LIN {X 0,Y 375.701,Z 668.969,A -85,B 0,C 180,E1 9709.263,E2 9709.263} C_VEL
LIN {X 0,Y 377.557,Z 672.937,A -85,B 0,C 180,E1 9707.734,E2 9707.734} C_VEL
LIN {X 0,Y 377.796,Z 674.692,A -85,B 0,C 180,E1 9707.454,E2 9707.454} C_VEL
LIN {X 0,Y 377.643,Z 677.934,A -85,B 0,C 180,E1 9707.299,E2 9707.299} C_VEL
LIN {X 0,Y 376.937,Z 683.014,A -85,B 0,C 180,E1 9707.331,E2 9707.331} C_VEL
LIN {X 0,Y 374.94,Z 694.139,A -85,B 0,C 180,E1 9707.675,E2 9707.675} C_VEL
LIN {X 0,Y 374.614,Z 696.752,A -85,B 0,C 180,E1 9707.671,E2 9707.671} C_VEL
LIN {X 0,Y 359.205,Z 844.41,A -85,B 0,C 180,E1 9705.429,E2 9705.429} C_VEL
LIN {X 0,Y 354.864,Z 869.774,A -85,B 0,C 180,E1 9704.944,E2 9704.944} C_VEL
LIN {X 0,Y 349.639,Z 892.086,A -85,B 0,C 180,E1 9704.392,E2 9704.392} C_VEL
LIN {X 0,Y 342.832,Z 914.874,A -85,B 0,C 180,E1 9703.649,E2 9703.649} C_VEL
LIN {X 0,Y 335.898,Z 934.267,A -85,B 0,C 180,E1 9702.852,E2 9702.852} C_VEL
LIN {X 0,Y 326.048,Z 957.663,A -85,B 0,C 180,E1 9701.649,E2 9701.649} C_VEL
LIN {X 0,Y 316.768,Z 976.66,A -85,B 0,C 180,E1 9700.43,E2 9700.43} C_VEL
LIN {X 0,Y 304.761,Z 998.24,A -85,B 0,C 180,E1 9698.714,E2 9698.714} C_VEL
LIN {X 0,Y 293.47,Z 1016.27,A -85,B 0,C 180,E1 9696.916,E2 9696.916} C_VEL
LIN {X 0,Y 279.783,Z 1035.844,A -85,B 0,C 180,E1 9694.474,E2 9694.474} C_VEL
LIN {X 0,Y 267.39,Z 1051.959,A -85,B 0,C 180,E1 9691.947,E2 9691.947} C_VEL
LIN {X 0,Y 253.812,Z 1068.099,A -85,B 0,C 180,E1 9688.746,E2 9688.746} C_VEL
LIN {X 0,Y 241.74,Z 1081.488,A -85,B 0,C 180,E1 9685.398,E2 9685.398} C_VEL
LIN {X 0,Y 228.302,Z 1095.466,A -85,B 0,C 180,E1 9680.9,E2 9680.9} C_VEL
LIN {X 0,Y 217.176,Z 1106.587,A -85,B 0,C 180,E1 9676.29,E2 9676.29} C_VEL
LIN {X 0,Y 206.281,Z 1117.208,A -85,B 0,C 180,E1 9670.506,E2 9670.506} C_VEL
LIN {X 0,Y 197.909,Z 1125.557,A -85,B 0,C 180,E1 9664.561,E2 9664.561} C_VEL
LIN {X 0,Y 191.158,Z 1132.65,A -85,B 0,C 180,E1 9657.745,E2 9657.745} C_VEL
LIN {X 0,Y 187.088,Z 1137.624,A -85,B 0,C 180,E1 9651.311,E2 9651.311} C_VEL
LIN {X 0,Y 184.611,Z 1141.644,A -85,B 0,C 180,E1 9643.787,E2 9643.787} C_VEL
LIN {X 0,Y 183.999,Z 1143.579,A -85,B 0,C 180,E1 9637.808,E2 9637.808} C_VEL
LIN {X 0,Y 183.993,Z 1144.393,A -85,B 0,C 180,E1 9632.803,E2 9632.803} C_VEL
LIN {X 0,Y 184.01,Z 1144.46,A -85,B 0,C 180,E1 9628.132,E2 9628.132} C_VEL
LIN {X 0,Y 184,Z 1143.707,A -85,B 0,C 180,E1 9622.82,E2 9622.82} C_VEL
LIN {X 0,Y 184.451,Z 1141.975,A -85,B 0,C 180,E1 9617.158,E2 9617.158} C_VEL
LIN {X 0,Y 186.519,Z 1138.434,A -85,B 0,C 180,E1 9609.935,E2 9609.935} C_VEL
LIN {X 0,Y 190.686,Z 1133.117,A -85,B 0,C 180,E1 9602.858,E2 9602.858} C_VEL
LIN {X 0,Y 197.142,Z 1126.294,A -85,B 0,C 180,E1 9596.088,E2 9596.088} C_VEL
LIN {X 0,Y 205.419,Z 1117.938,A -85,B 0,C 180,E1 9590.02,E2 9590.02} C_VEL
LIN {X 0,Y 215.636,Z 1108.026,A -85,B 0,C 180,E1 9584.431,E2 9584.431} C_VEL
LIN {X 0,Y 227.015,Z 1096.607,A -85,B 0,C 180,E1 9579.575,E2 9579.575} C_VEL
LIN {X 0,Y 239.804,Z 1083.447,A -85,B 0,C 180,E1 9575.19,E2 9575.19} C_VEL
LIN {X 0,Y 252.416,Z 1069.461,A -85,B 0,C 180,E1 9571.605,E2 9571.605} C_VEL
LIN {X 0,Y 265.911,Z 1053.589,A -85,B 0,C 180,E1 9568.369,E2 9568.369} C_VEL
LIN {X 0,Y 278.635,Z 1037.085,A -85,B 0,C 180,E1 9565.735,E2 9565.735} C_VEL
LIN {X 0,Y 291.47,Z 1019.01,A -85,B 0,C 180,E1 9563.413,E2 9563.413} C_VEL
LIN {X 0,Y 303.11,Z 1000.561,A -85,B 0,C 180,E1 9561.525,E2 9561.525} C_VEL
LIN {X 0,Y 314.301,Z 981.008,A -85,B 0,C 180,E1 9559.901,E2 9559.901} C_VEL
LIN {X 0,Y 324.332,Z 960.785,A -85,B 0,C 180,E1 9558.558,E2 9558.558} C_VEL
LIN {X 0,Y 333.728,Z 939.306,A -85,B 0,C 180,E1 9557.394,E2 9557.394} C_VEL
LIN {X 0,Y 341.5,Z 918.015,A -85,B 0,C 180,E1 9556.483,E2 9556.483} C_VEL
LIN {X 0,Y 348.715,Z 894.664,A -85,B 0,C 180,E1 9555.694,E2 9555.694} C_VEL
LIN {X 0,Y 354.348,Z 870.929,A -85,B 0,C 180,E1 9555.095,E2 9555.095} C_VEL
LIN {X 0,Y 358.67,Z 846.5,A -85,B 0,C 180,E1 9554.619,E2 9554.619} C_VEL
LIN {X 0,Y 365.964,Z 777.896,A -85,B 0,C 180,E1 9553.555,E2 9553.555} C_VEL
LIN {X 0,Y 375.97,Z 680.709,A -85,B 0,C 180,E1 9552.089,E2 9552.089} C_VEL
LIN {X 0,Y 373.012,Z 674.26,A -85,B 0,C 180,E1 9549.489,E2 9549.489} C_VEL
LIN {X 0,Y 370.608,Z 669.322,A -85,B 0,C 180,E1 9546.818,E2 9546.818} C_VEL
LIN {X 0,Y 369.056,Z 666.191,A -85,B 0,C 180,E1 9544.506,E2 9544.506} C_VEL
LIN {X 0,Y 367.518,Z 663.322,A -85,B 0,C 180,E1 9540.624,E2 9540.624} C_VEL
LIN {X 0,Y 367.214,Z 663.186,A -85,B 0,C 180,E1 9538.284,E2 9538.284} C_VEL
LIN {X 0,Y 368.066,Z 666.012,A -85,B 0,C 180,E1 9533.605,E2 9533.605} C_VEL
LIN {X 0,Y 369.73,Z 670.596,A -85,B 0,C 180,E1 9530.426,E2 9530.426} C_VEL
LIN {X 0,Y 372.279,Z 677.037,A -85,B 0,C 180,E1 9527.316,E2 9527.316} C_VEL
LIN {X 0,Y 375.214,Z 684.89,A -85,B 0,C 180,E1 9524.564,E2 9524.564} C_VEL
LIN {X 0,Y 358.827,Z 845.607,A -85,B 0,C 180,E1 9522.185,E2 9522.185} C_VEL
LIN {X 0,Y 354.604,Z 870.442,A -85,B 0,C 180,E1 9521.723,E2 9521.723} C_VEL
LIN {X 0,Y 349.339,Z 892.966,A -85,B 0,C 180,E1 9521.175,E2 9521.175} C_VEL
LIN {X 0,Y 342.711,Z 915.03,A -85,B 0,C 180,E1 9520.456,E2 9520.456} C_VEL
LIN {X 0,Y 335.451,Z 935.225,A -85,B 0,C 180,E1 9519.627,E2 9519.627} C_VEL
LIN {X 0,Y 326.046,Z 957.24,A -85,B 0,C 180,E1 9518.487,E2 9518.487} C_VEL
LIN {X 0,Y 317.01,Z 975.595,A -85,B 0,C 180,E1 9517.308,E2 9517.308} C_VEL
LIN {X 0,Y 305.169,Z 996.623,A -85,B 0,C 180,E1 9515.627,E2 9515.627} C_VEL
LIN {X 0,Y 294.024,Z 1014.21,A -85,B 0,C 180,E1 9513.87,E2 9513.87} C_VEL
LIN {X 0,Y 281.274,Z 1032.172,A -85,B 0,C 180,E1 9511.622,E2 9511.622} C_VEL
LIN {X 0,Y 268.993,Z 1047.885,A -85,B 0,C 180,E1 9509.168,E2 9509.168} C_VEL
LIN {X 0,Y 255.516,Z 1063.539,A -85,B 0,C 180,E1 9506.058,E2 9506.058} C_VEL
LIN {X 0,Y 242.86,Z 1077.178,A -85,B 0,C 180,E1 9502.619,E2 9502.619} C_VEL
LIN {X 0,Y 230.542,Z 1089.435,A -85,B 0,C 180,E1 9498.619,E2 9498.619} C_VEL
LIN {X 0,Y 218.914,Z 1100.521,A -85,B 0,C 180,E1 9493.969,E2 9493.969} C_VEL
LIN {X 0,Y 208.319,Z 1110.115,A -85,B 0,C 180,E1 9488.607,E2 9488.607} C_VEL
LIN {X 0,Y 199.344,Z 1118.32,A -85,B 0,C 180,E1 9482.576,E2 9482.576} C_VEL
LIN {X 0,Y 192.297,Z 1124.808,A -85,B 0,C 180,E1 9475.899,E2 9475.899} C_VEL
LIN {X 0,Y 187.614,Z 1129.68,A -85,B 0,C 180,E1 9468.972,E2 9468.972} C_VEL
LIN {X 0,Y 185.097,Z 1132.745,A -85,B 0,C 180,E1 9462.105,E2 9462.105} C_VEL
LIN {X 0,Y 184.194,Z 1134.377,A -85,B 0,C 180,E1 9455.92,E2 9455.92} C_VEL
LIN {X 0,Y 184.04,Z 1134.934,A -85,B 0,C 180,E1 9449.689,E2 9449.689} C_VEL
LIN {X 0,Y 184.237,Z 1134.282,A -85,B 0,C 180,E1 9443.456,E2 9443.456} C_VEL
LIN {X 0,Y 185.163,Z 1132.676,A -85,B 0,C 180,E1 9437.526,E2 9437.526} C_VEL
LIN {X 0,Y 187.925,Z 1129.387,A -85,B 0,C 180,E1 9430.351,E2 9430.351} C_VEL
LIN {X 0,Y 192.747,Z 1124.444,A -85,B 0,C 180,E1 9423.504,E2 9423.504} C_VEL
LIN {X 0,Y 199.846,Z 1117.935,A -85,B 0,C 180,E1 9416.95,E2 9416.95} C_VEL
LIN {X 0,Y 208.659,Z 1109.922,A -85,B 0,C 180,E1 9411.115,E2 9411.115} C_VEL
LIN {X 0,Y 219.841,Z 1099.761,A -85,B 0,C 180,E1 9405.538,E2 9405.538} C_VEL
LIN {X 0,Y 231.005,Z 1089.152,A -85,B 0,C 180,E1 9401.136,E2 9401.136} C_VEL
LIN {X 0,Y 244.665,Z 1075.45,A -85,B 0,C 180,E1 9396.773,E2 9396.773} C_VEL
LIN {X 0,Y 256.763,Z 1062.396,A -85,B 0,C 180,E1 9393.554,E2 9393.554} C_VEL
LIN {X 0,Y 270.582,Z 1046.165,A -85,B 0,C 180,E1 9390.415,E2 9390.415} C_VEL
LIN {X 0,Y 282.352,Z 1031.055,A -85,B 0,C 180,E1 9388.099,E2 9388.099} C_VEL
LIN {X 0,Y 295.457,Z 1012.382,A -85,B 0,C 180,E1 9385.815,E2 9385.815} C_VEL
LIN {X 0,Y 306.65,Z 994.615,A -85,B 0,C 180,E1 9384.077,E2 9384.077} C_VEL
LIN {X 0,Y 318.112,Z 973.95,A -85,B 0,C 180,E1 9382.466,E2 9382.466} C_VEL
LIN {X 0,Y 327.706,Z 954.261,A -85,B 0,C 180,E1 9381.229,E2 9381.229} C_VEL
LIN {X 0,Y 336.673,Z 932.69,A -85,B 0,C 180,E1 9380.152,E2 9380.152} C_VEL
LIN {X 0,Y 343.874,Z 912.39,A -85,B 0,C 180,E1 9379.342,E2 9379.342} C_VEL
LIN {X 0,Y 350.593,Z 889.059,A -85,B 0,C 180,E1 9378.618,E2 9378.618} C_VEL
LIN {X 0,Y 355.597,Z 867.034,A -85,B 0,C 180,E1 9378.102,E2 9378.102} C_VEL
LIN {X 0,Y 359.466,Z 842.639,A -85,B 0,C 180,E1 9377.665,E2 9377.665} C_VEL
LIN {X 0,Y 375.46,Z 685.049,A -85,B 0,C 180,E1 9375.322,E2 9375.322} C_VEL
LIN {X 0,Y 372.379,Z 676.838,A -85,B 0,C 180,E1 9372.405,E2 9372.405} C_VEL
LIN {X 0,Y 369.893,Z 670.489,A -85,B 0,C 180,E1 9369.256,E2 9369.256} C_VEL
LIN {X 0,Y 368.194,Z 665.764,A -85,B 0,C 180,E1 9365.767,E2 9365.767} C_VEL
LIN {X 0,Y 367.559,Z 663.495,A -85,B 0,C 180,E1 9361.091,E2 9361.091} C_VEL
LIN {X 0,Y 368.011,Z 664.084,A -85,B 0,C 180,E1 9358.599,E2 9358.599} C_VEL
LIN {X 0,Y 369.718,Z 667.153,A -85,B 0,C 180,E1 9354.88,E2 9354.88} C_VEL
LIN {X 0,Y 371.838,Z 671.522,A -85,B 0,C 180,E1 9352.04,E2 9352.04} C_VEL
LIN {X 0,Y 374.332,Z 676.68,A -85,B 0,C 180,E1 9349.535,E2 9349.535} C_VEL
LIN {X 0,Y 376.229,Z 681.199,A -85,B 0,C 180,E1 9347.901,E2 9347.901} C_VEL
LIN {X 0,Y 374.614,Z 696.752,A -85,B 0,C 180,E1 9347.671,E2 9347.671} C_VEL
LIN {X 0,Y 373.569,Z 704.446,A -85,B 0,C 180,E1 9347.707,E2 9347.707} C_VEL
LIN {X 0,Y 369.939,Z 724.972,A -85,B 0,C 180,E1 9348.345,E2 9348.345} C_VEL
LIN {X 0,Y 369.073,Z 731.573,A -85,B 0,C 180,E1 9348.36,E2 9348.36} C_VEL
LIN {X 0,Y 357.006,Z 844.853,A -85,B 0,C 180,E1 9346.658,E2 9346.658} C_VEL
LIN {X 0,Y 352.627,Z 869.936,A -85,B 0,C 180,E1 9346.19,E2 9346.19} C_VEL
LIN {X 0,Y 347.283,Z 892.401,A -85,B 0,C 180,E1 9345.649,E2 9345.649} C_VEL
LIN {X 0,Y 340.08,Z 915.965,A -85,B 0,C 180,E1 9344.898,E2 9344.898} C_VEL
LIN {X 0,Y 332.72,Z 936.065,A -85,B 0,C 180,E1 9344.085,E2 9344.085} C_VEL
LIN {X 0,Y 323.145,Z 958.179,A -85,B 0,C 180,E1 9342.965,E2 9342.965} C_VEL
LIN {X 0,Y 313.279,Z 977.938,A -85,B 0,C 180,E1 9341.72,E2 9341.72} C_VEL
LIN {X 0,Y 301.054,Z 999.277,A -85,B 0,C 180,E1 9340.04,E2 9340.04} C_VEL
LIN {X 0,Y 289.54,Z 1017.204,A -85,B 0,C 180,E1 9338.274,E2 9338.274} C_VEL
LIN {X 0,Y 275.944,Z 1036.087,A -85,B 0,C 180,E1 9335.942,E2 9335.942} C_VEL
LIN {X 0,Y 263.611,Z 1051.698,A -85,B 0,C 180,E1 9333.53,E2 9333.53} C_VEL
LIN {X 0,Y 249.62,Z 1067.856,A -85,B 0,C 180,E1 9330.369,E2 9330.369} C_VEL
LIN {X 0,Y 237.131,Z 1081.249,A -85,B 0,C 180,E1 9327.046,E2 9327.046} C_VEL
LIN {X 0,Y 223.656,Z 1094.763,A -85,B 0,C 180,E1 9322.729,E2 9322.729} C_VEL
LIN {X 0,Y 212.066,Z 1105.833,A -85,B 0,C 180,E1 9318.157,E2 9318.157} C_VEL
LIN {X 0,Y 200.5,Z 1116.571,A -85,B 0,C 180,E1 9312.318,E2 9312.318} C_VEL
LIN {X 0,Y 191.77,Z 1124.712,A -85,B 0,C 180,E1 9306.47,E2 9306.47} C_VEL
LIN {X 0,Y 184.148,Z 1132.17,A -85,B 0,C 180,E1 9299.254,E2 9299.254} C_VEL
LIN {X 0,Y 179.628,Z 1137.193,A -85,B 0,C 180,E1 9292.587,E2 9292.587} C_VEL
LIN {X 0,Y 176.786,Z 1141.319,A -85,B 0,C 180,E1 9284.722,E2 9284.722} C_VEL
LIN {X 0,Y 176.01,Z 1143.368,A -85,B 0,C 180,E1 9278.165,E2 9278.165} C_VEL
LIN {X 0,Y 175.994,Z 1144.183,A -85,B 0,C 180,E1 9272.931,E2 9272.931} C_VEL
LIN {X 0,Y 176.01,Z 1144.25,A -85,B 0,C 180,E1 9268.047,E2 9268.047} C_VEL
LIN {X 0,Y 176.001,Z 1143.568,A -85,B 0,C 180,E1 9262.82,E2 9262.82} C_VEL
LIN {X 0,Y 176.481,Z 1141.881,A -85,B 0,C 180,E1 9256.901,E2 9256.901} C_VEL
LIN {X 0,Y 178.418,Z 1138.742,A -85,B 0,C 180,E1 9250.01,E2 9250.01} C_VEL
LIN {X 0,Y 182.894,Z 1133.424,A -85,B 0,C 180,E1 9242.309,E2 9242.309} C_VEL
LIN {X 0,Y 188.94,Z 1127.333,A -85,B 0,C 180,E1 9235.877,E2 9235.877} C_VEL
LIN {X 0,Y 198.247,Z 1118.544,A -85,B 0,C 180,E1 9229.029,E2 9229.029} C_VEL
LIN {X 0,Y 207.807,Z 1109.679,A -85,B 0,C 180,E1 9223.801,E2 9223.801} C_VEL
LIN {X 0,Y 220.623,Z 1097.543,A -85,B 0,C 180,E1 9218.366,E2 9218.366} C_VEL
LIN {X 0,Y 232.489,Z 1085.818,A -85,B 0,C 180,E1 9214.334,E2 9214.334} C_VEL
LIN {X 0,Y 246.765,Z 1070.777,A -85,B 0,C 180,E1 9210.336,E2 9210.336} C_VEL
LIN {X 0,Y 259.098,Z 1056.809,A -85,B 0,C 180,E1 9207.427,E2 9207.427} C_VEL
LIN {X 0,Y 273.581,Z 1038.886,A -85,B 0,C 180,E1 9204.487,E2 9204.487} C_VEL
LIN {X 0,Y 285.48,Z 1022.721,A -85,B 0,C 180,E1 9202.383,E2 9202.383} C_VEL
LIN {X 0,Y 298.547,Z 1002.939,A -85,B 0,C 180,E1 9200.318,E2 9200.318} C_VEL
LIN {X 0,Y 309.019,Z 985.235,A -85,B 0,C 180,E1 9198.836,E2 9198.836} C_VEL
LIN {X 0,Y 320.542,Z 963.106,A -85,B 0,C 180,E1 9197.343,E2 9197.343} C_VEL
LIN {X 0,Y 329.2,Z 943.943,A -85,B 0,C 180,E1 9196.3,E2 9196.3} C_VEL
LIN {X 0,Y 338.406,Z 920.041,A -85,B 0,C 180,E1 9195.265,E2 9195.265} C_VEL
LIN {X 0,Y 345.052,Z 899.254,A -85,B 0,C 180,E1 9194.564,E2 9194.564} C_VEL
LIN {X 0,Y 351.521,Z 873.81,A -85,B 0,C 180,E1 9193.908,E2 9193.908} C_VEL
LIN {X 0,Y 355.776,Z 851.301,A -85,B 0,C 180,E1 9193.466,E2 9193.466} C_VEL
LIN {X 0,Y 359.782,Z 817.87,A -85,B 0,C 180,E1 9192.936,E2 9192.936} C_VEL
LIN {X 0,Y 373.543,Z 686.091,A -85,B 0,C 180,E1 9190.956,E2 9190.956} C_VEL
LIN {X 0,Y 370.614,Z 679.643,A -85,B 0,C 180,E1 9188.065,E2 9188.065} C_VEL
LIN {X 0,Y 369.036,Z 676.353,A -85,B 0,C 180,E1 9186.066,E2 9186.066} C_VEL
LIN {X 0,Y 367.984,Z 674.066,A -85,B 0,C 180,E1 9184.363,E2 9184.363} C_VEL
LIN {X 0,Y 366.509,Z 671.213,A -85,B 0,C 180,E1 9180.469,E2 9180.469} C_VEL
LIN {X 0,Y 366.233,Z 671.188,A -85,B 0,C 180,E1 9178.122,E2 9178.122} C_VEL
LIN {X 0,Y 367.02,Z 673.937,A -85,B 0,C 180,E1 9173.744,E2 9173.744} C_VEL
LIN {X 0,Y 368.587,Z 678.422,A -85,B 0,C 180,E1 9170.632,E2 9170.632} C_VEL
LIN {X 0,Y 370.912,Z 684.617,A -85,B 0,C 180,E1 9167.664,E2 9167.664} C_VEL
LIN {X 0,Y 372.841,Z 690.31,A -85,B 0,C 180,E1 9165.682,E2 9165.682} C_VEL
LIN {X 0,Y 356.687,Z 845.48,A -85,B 0,C 180,E1 9163.423,E2 9163.423} C_VEL
LIN {X 0,Y 352.383,Z 870.437,A -85,B 0,C 180,E1 9162.971,E2 9162.971} C_VEL
LIN {X 0,Y 347.07,Z 892.849,A -85,B 0,C 180,E1 9162.443,E2 9162.443} C_VEL
LIN {X 0,Y 340.123,Z 915.582,A -85,B 0,C 180,E1 9161.724,E2 9161.724} C_VEL
LIN {X 0,Y 332.752,Z 935.713,A -85,B 0,C 180,E1 9160.918,E2 9160.918} C_VEL
LIN {X 0,Y 323.453,Z 957.092,A -85,B 0,C 180,E1 9159.84,E2 9159.84} C_VEL
LIN {X 0,Y 313.999,Z 975.96,A -85,B 0,C 180,E1 9158.659,E2 9158.659} C_VEL
LIN {X 0,Y 301.936,Z 996.938,A -85,B 0,C 180,E1 9157.018,E2 9157.018} C_VEL
LIN {X 0,Y 290.559,Z 1014.508,A -85,B 0,C 180,E1 9155.299,E2 9155.299} C_VEL
LIN {X 0,Y 277.52,Z 1032.443,A -85,B 0,C 180,E1 9153.092,E2 9153.092} C_VEL
LIN {X 0,Y 264.928,Z 1048.146,A -85,B 0,C 180,E1 9150.674,E2 9150.674} C_VEL
LIN {X 0,Y 251.069,Z 1063.785,A -85,B 0,C 180,E1 9147.597,E2 9147.597} C_VEL
LIN {X 0,Y 238.007,Z 1077.418,A -85,B 0,C 180,E1 9144.176,E2 9144.176} C_VEL
LIN {X 0,Y 225.235,Z 1089.663,A -85,B 0,C 180,E1 9140.175,E2 9140.175} C_VEL
LIN {X 0,Y 213.657,Z 1100.242,A -85,B 0,C 180,E1 9135.728,E2 9135.728} C_VEL
LIN {X 0,Y 202.468,Z 1109.939,A -85,B 0,C 180,E1 9130.312,E2 9130.312} C_VEL
LIN {X 0,Y 193.141,Z 1117.975,A -85,B 0,C 180,E1 9124.353,E2 9124.353} C_VEL
LIN {X 0,Y 185.556,Z 1124.53,A -85,B 0,C 180,E1 9117.608,E2 9117.608} C_VEL
LIN {X 0,Y 180.308,Z 1129.536,A -85,B 0,C 180,E1 9110.448,E2 9110.448} C_VEL
LIN {X 0,Y 177.312,Z 1132.828,A -85,B 0,C 180,E1 9103.036,E2 9103.036} C_VEL
LIN {X 0,Y 176.266,Z 1134.457,A -85,B 0,C 180,E1 9096.842,E2 9096.842} C_VEL
LIN {X 0,Y 176.047,Z 1135.132,A -85,B 0,C 180,E1 9090.325,E2 9090.325} C_VEL
LIN {X 0,Y 176.21,Z 1134.623,A -85,B 0,C 180,E1 9083.811,E2 9083.811} C_VEL
LIN {X 0,Y 177.205,Z 1132.996,A -85,B 0,C 180,E1 9077.287,E2 9077.287} C_VEL
LIN {X 0,Y 180.089,Z 1129.82,A -85,B 0,C 180,E1 9069.865,E2 9069.865} C_VEL
LIN {X 0,Y 185.214,Z 1124.905,A -85,B 0,C 180,E1 9062.685,E2 9062.685} C_VEL
LIN {X 0,Y 192.679,Z 1118.493,A -85,B 0,C 180,E1 9055.912,E2 9055.912} C_VEL
LIN {X 0,Y 202.365,Z 1110.14,A -85,B 0,C 180,E1 9049.663,E2 9049.663} C_VEL
LIN {X 0,Y 214.088,Z 1099.984,A -85,B 0,C 180,E1 9044.007,E2 9044.007} C_VEL
LIN {X 0,Y 225.724,Z 1089.376,A -85,B 0,C 180,E1 9039.577,E2 9039.577} C_VEL
LIN {X 0,Y 239.88,Z 1075.684,A -85,B 0,C 180,E1 9035.215,E2 9035.215} C_VEL
LIN {X 0,Y 252.36,Z 1062.634,A -85,B 0,C 180,E1 9032.015,E2 9032.015} C_VEL
LIN {X 0,Y 266.293,Z 1046.756,A -85,B 0,C 180,E1 9028.969,E2 9028.969} C_VEL
LIN {X 0,Y 278.555,Z 1031.418,A -85,B 0,C 180,E1 9026.645,E2 9026.645} C_VEL
LIN {X 0,Y 292.033,Z 1012.673,A -85,B 0,C 180,E1 9024.389,E2 9024.389} C_VEL
LIN {X 0,Y 303.454,Z 994.922,A -85,B 0,C 180,E1 9022.689,E2 9022.689} C_VEL
LIN {X 0,Y 315.131,Z 974.305,A -85,B 0,C 180,E1 9021.117,E2 9021.117} C_VEL
LIN {X 0,Y 324.889,Z 954.646,A -85,B 0,C 180,E1 9019.911,E2 9019.911} C_VEL
LIN {X 0,Y 334.014,Z 933.135,A -85,B 0,C 180,E1 9018.863,E2 9018.863} C_VEL
LIN {X 0,Y 341.269,Z 913.053,A -85,B 0,C 180,E1 9018.081,E2 9018.081} C_VEL
LIN {X 0,Y 348.28,Z 889.203,A -85,B 0,C 180,E1 9017.36,E2 9017.36} C_VEL
LIN {X 0,Y 353.371,Z 867.137,A -85,B 0,C 180,E1 9016.859,E2 9016.859} C_VEL
LIN {X 0,Y 357.33,Z 842.607,A -85,B 0,C 180,E1 9016.429,E2 9016.429} C_VEL
LIN {X 0,Y 373.1,Z 690.229,A -85,B 0,C 180,E1 9014.195,E2 9014.195} C_VEL
LIN {X 0,Y 370.431,Z 682.823,A -85,B 0,C 180,E1 9011.364,E2 9011.364} C_VEL
LIN {X 0,Y 368.48,Z 677.548,A -85,B 0,C 180,E1 9008.583,E2 9008.583} C_VEL
LIN {X 0,Y 367.113,Z 673.554,A -85,B 0,C 180,E1 9005.47,E2 9005.47} C_VEL
LIN {X 0,Y 366.583,Z 671.437,A -85,B 0,C 180,E1 9001.094,E2 9001.094} C_VEL
LIN {X 0,Y 367.023,Z 672.068,A -85,B 0,C 180,E1 8998.595,E2 8998.595} C_VEL
LIN {X 0,Y 368.625,Z 675.066,A -85,B 0,C 180,E1 8995.02,E2 8995.02} C_VEL
LIN {X 0,Y 370.568,Z 679.204,A -85,B 0,C 180,E1 8992.324,E2 8992.324} C_VEL
LIN {X 0,Y 372.89,Z 684.225,A -85,B 0,C 180,E1 8989.884,E2 8989.884} C_VEL
LIN {X 0,Y 373.813,Z 686.677,A -85,B 0,C 180,E1 8989.013,E2 8989.013} C_VEL
LIN {X 0,Y 369.073,Z 731.573,A -85,B 0,C 180,E1 8988.36,E2 8988.36} C_VEL
LIN {X 0,Y 368.033,Z 739.267,A -85,B 0,C 180,E1 8988.399,E2 8988.399} C_VEL
LIN {X 0,Y 364.446,Z 759.789,A -85,B 0,C 180,E1 8989.058,E2 8989.058} C_VEL
LIN {X 0,Y 363.586,Z 766.389,A -85,B 0,C 180,E1 8989.073,E2 8989.073} C_VEL
LIN {X 0,Y 354.933,Z 845.615,A -85,B 0,C 180,E1 8987.896,E2 8987.896} C_VEL
LIN {X 0,Y 350.516,Z 870.293,A -85,B 0,C 180,E1 8987.446,E2 8987.446} C_VEL
LIN {X 0,Y 344.987,Z 893.137,A -85,B 0,C 180,E1 8986.912,E2 8986.912} C_VEL
LIN {X 0,Y 337.729,Z 916.376,A -85,B 0,C 180,E1 8986.19,E2 8986.19} C_VEL
LIN {X 0,Y 329.699,Z 937.863,A -85,B 0,C 180,E1 8985.341,E2 8985.341} C_VEL
LIN {X 0,Y 319.977,Z 959.603,A -85,B 0,C 180,E1 8984.253,E2 8984.253} C_VEL
LIN {X 0,Y 309.522,Z 980.035,A -85,B 0,C 180,E1 8982.982,E2 8982.982} C_VEL
LIN {X 0,Y 297.511,Z 1000.314,A -85,B 0,C 180,E1 8981.399,E2 8981.399} C_VEL
LIN {X 0,Y 284.95,Z 1019.364,A -85,B 0,C 180,E1 8979.538,E2 8979.538} C_VEL
LIN {X 0,Y 271.489,Z 1037.358,A -85,B 0,C 180,E1 8977.308,E2 8977.308} C_VEL
LIN {X 0,Y 257.723,Z 1054.217,A -85,B 0,C 180,E1 8974.686,E2 8974.686} C_VEL
LIN {X 0,Y 243.646,Z 1069.732,A -85,B 0,C 180,E1 8971.572,E2 8971.572} C_VEL
LIN {X 0,Y 229.291,Z 1084.458,A -85,B 0,C 180,E1 8967.779,E2 8967.779} C_VEL
LIN {X 0,Y 216.208,Z 1096.873,A -85,B 0,C 180,E1 8963.581,E2 8963.581} C_VEL
LIN {X 0,Y 203.194,Z 1108.679,A -85,B 0,C 180,E1 8958.37,E2 8958.37} C_VEL
LIN {X 0,Y 192.535,Z 1118.01,A -85,B 0,C 180,E1 8952.869,E2 8952.869} C_VEL
LIN {X 0,Y 182.883,Z 1126.566,A -85,B 0,C 180,E1 8946.191,E2 8946.191} C_VEL
LIN {X 0,Y 175.894,Z 1133.006,A -85,B 0,C 180,E1 8939.267,E2 8939.267} C_VEL
LIN {X 0,Y 171.05,Z 1138.232,A -85,B 0,C 180,E1 8931.609,E2 8931.609} C_VEL
LIN {X 0,Y 168.635,Z 1141.576,A -85,B 0,C 180,E1 8924.07,E2 8924.07} C_VEL
LIN {X 0,Y 168.002,Z 1143.301,A -85,B 0,C 180,E1 8917.868,E2 8917.868} C_VEL
LIN {X 0,Y 168.004,Z 1144.021,A -85,B 0,C 180,E1 8912.388,E2 8912.388} C_VEL
LIN {X 0,Y 168.004,Z 1144.016,A -85,B 0,C 180,E1 8907.612,E2 8907.612} C_VEL
LIN {X 0,Y 168.005,Z 1143.284,A -85,B 0,C 180,E1 8902.132,E2 8902.132} C_VEL
LIN {X 0,Y 168.635,Z 1141.548,A -85,B 0,C 180,E1 8895.93,E2 8895.93} C_VEL
LIN {X 0,Y 171.208,Z 1137.999,A -85,B 0,C 180,E1 8888.051,E2 8888.051} C_VEL
LIN {X 0,Y 176.157,Z 1132.678,A -85,B 0,C 180,E1 8880.408,E2 8880.408} C_VEL
LIN {X 0,Y 183.692,Z 1125.785,A -85,B 0,C 180,E1 8873.146,E2 8873.146} C_VEL
LIN {X 0,Y 193.472,Z 1117.075,A -85,B 0,C 180,E1 8866.578,E2 8866.578} C_VEL
LIN {X 0,Y 205.033,Z 1106.942,A -85,B 0,C 180,E1 8860.805,E2 8860.805} C_VEL
LIN {X 0,Y 217.45,Z 1095.554,A -85,B 0,C 180,E1 8855.973,E2 8855.973} C_VEL
LIN {X 0,Y 231.332,Z 1082.246,A -85,B 0,C 180,E1 8851.624,E2 8851.624} C_VEL
LIN {X 0,Y 244.885,Z 1068.18,A -85,B 0,C 180,E1 8848.121,E2 8848.121} C_VEL
LIN {X 0,Y 259.249,Z 1052.117,A -85,B 0,C 180,E1 8844.991,E2 8844.991} C_VEL
LIN {X 0,Y 272.217,Z 1036.117,A -85,B 0,C 180,E1 8842.552,E2 8842.552} C_VEL
LIN {X 0,Y 285.758,Z 1017.785,A -85,B 0,C 180,E1 8840.322,E2 8840.322} C_VEL
LIN {X 0,Y 297.492,Z 999.917,A -85,B 0,C 180,E1 8838.59,E2 8838.59} C_VEL
LIN {X 0,Y 309.502,Z 979.549,A -85,B 0,C 180,E1 8837.006,E2 8837.006} C_VEL
LIN {X 0,Y 319.655,Z 959.701,A -85,B 0,C 180,E1 8835.771,E2 8835.771} C_VEL
LIN {X 0,Y 329.205,Z 938.415,A -85,B 0,C 180,E1 8834.699,E2 8834.699} C_VEL
LIN {X 0,Y 337.262,Z 916.897,A -85,B 0,C 180,E1 8833.843,E2 8833.843} C_VEL
LIN {X 0,Y 344.576,Z 893.611,A -85,B 0,C 180,E1 8833.114,E2 8833.114} C_VEL
LIN {X 0,Y 350.172,Z 870.54,A -85,B 0,C 180,E1 8832.571,E2 8832.571} C_VEL
LIN {X 0,Y 354.603,Z 845.902,A -85,B 0,C 180,E1 8832.121,E2 8832.121} C_VEL
LIN {X 0,Y 363.543,Z 764.207,A -85,B 0,C 180,E1 8830.905,E2 8830.905} C_VEL
LIN {X 0,Y 371.28,Z 691.711,A -85,B 0,C 180,E1 8829.847,E2 8829.847} C_VEL
LIN {X 0,Y 368.831,Z 686.149,A -85,B 0,C 180,E1 8827.151,E2 8827.151} C_VEL
LIN {X 0,Y 366.915,Z 681.941,A -85,B 0,C 180,E1 8824.22,E2 8824.22} C_VEL
LIN {X 0,Y 365.502,Z 679.106,A -85,B 0,C 180,E1 8820.313,E2 8820.313} C_VEL
LIN {X 0,Y 365.252,Z 679.205,A -85,B 0,C 180,E1 8817.961,E2 8817.961} C_VEL
LIN {X 0,Y 365.976,Z 681.858,A -85,B 0,C 180,E1 8813.883,E2 8813.883} C_VEL
LIN {X 0,Y 367.448,Z 686.247,A -85,B 0,C 180,E1 8810.84,E2 8810.84} C_VEL
LIN {X 0,Y 369.555,Z 692.195,A -85,B 0,C 180,E1 8808.015,E2 8808.015} C_VEL
LIN {X 0,Y 370.623,Z 695.601,A -85,B 0,C 180,E1 8806.815,E2 8806.815} C_VEL
LIN {X 0,Y 354.676,Z 845.674,A -85,B 0,C 180,E1 8804.671,E2 8804.671} C_VEL
LIN {X 0,Y 350.33,Z 870.434,A -85,B 0,C 180,E1 8804.235,E2 8804.235} C_VEL
LIN {X 0,Y 344.945,Z 892.839,A -85,B 0,C 180,E1 8803.725,E2 8803.725} C_VEL
LIN {X 0,Y 337.705,Z 916.132,A -85,B 0,C 180,E1 8803.01,E2 8803.01} C_VEL
LIN {X 0,Y 329.547,Z 937.943,A -85,B 0,C 180,E1 8802.155,E2 8802.155} C_VEL
LIN {X 0,Y 320.201,Z 958.683,A -85,B 0,C 180,E1 8801.117,E2 8801.117} C_VEL
LIN {X 0,Y 309.892,Z 978.739,A -85,B 0,C 180,E1 8799.874,E2 8799.874} C_VEL
LIN {X 0,Y 298.376,Z 998.057,A -85,B 0,C 180,E1 8798.369,E2 8798.369} C_VEL
LIN {X 0,Y 286.059,Z 1016.613,A -85,B 0,C 180,E1 8796.57,E2 8796.57} C_VEL
LIN {X 0,Y 272.763,Z 1034.215,A -85,B 0,C 180,E1 8794.394,E2 8794.394} C_VEL
LIN {X 0,Y 259.527,Z 1050.22,A -85,B 0,C 180,E1 8791.919,E2 8791.919} C_VEL
LIN {X 0,Y 246.081,Z 1064.788,A -85,B 0,C 180,E1 8789.021,E2 8789.021} C_VEL
LIN {X 0,Y 232.652,Z 1078.344,A -85,B 0,C 180,E1 8785.607,E2 8785.607} C_VEL
LIN {X 0,Y 219.469,Z 1090.457,A -85,B 0,C 180,E1 8781.594,E2 8781.594} C_VEL
LIN {X 0,Y 206.908,Z 1101.471,A -85,B 0,C 180,E1 8776.863,E2 8776.863} C_VEL
LIN {X 0,Y 195.334,Z 1110.951,A -85,B 0,C 180,E1 8771.326,E2 8771.326} C_VEL
LIN {X 0,Y 185.227,Z 1119.189,A -85,B 0,C 180,E1 8764.862,E2 8764.862} C_VEL
LIN {X 0,Y 177.786,Z 1125.24,A -85,B 0,C 180,E1 8758.192,E2 8758.192} C_VEL
LIN {X 0,Y 172.346,Z 1130.106,A -85,B 0,C 180,E1 8750.726,E2 8750.726} C_VEL
LIN {X 0,Y 169.362,Z 1133.15,A -85,B 0,C 180,E1 8743.312,E2 8743.312} C_VEL
LIN {X 0,Y 168.238,Z 1134.799,A -85,B 0,C 180,E1 8736.484,E2 8736.484} C_VEL
LIN {X 0,Y 168.045,Z 1135.354,A -85,B 0,C 180,E1 8729.659,E2 8729.659} C_VEL
LIN {X 0,Y 168.293,Z 1134.703,A -85,B 0,C 180,E1 8722.833,E2 8722.833} C_VEL
LIN {X 0,Y 169.431,Z 1133.099,A -85,B 0,C 180,E1 8716.346,E2 8716.346} C_VEL
LIN {X 0,Y 172.68,Z 1129.854,A -85,B 0,C 180,E1 8708.605,E2 8708.605} C_VEL
LIN {X 0,Y 178.308,Z 1124.872,A -85,B 0,C 180,E1 8701.167,E2 8701.167} C_VEL
LIN {X 0,Y 186.373,Z 1118.37,A -85,B 0,C 180,E1 8694.212,E2 8694.212} C_VEL
LIN {X 0,Y 196.418,Z 1110.19,A -85,B 0,C 180,E1 8688.008,E2 8688.008} C_VEL
LIN {X 0,Y 208.497,Z 1100.207,A -85,B 0,C 180,E1 8682.393,E2 8682.393} C_VEL
LIN {X 0,Y 220.619,Z 1089.6,A -85,B 0,C 180,E1 8677.944,E2 8677.944} C_VEL
LIN {X 0,Y 235.279,Z 1075.917,A -85,B 0,C 180,E1 8673.595,E2 8673.595} C_VEL
LIN {X 0,Y 248.146,Z 1062.874,A -85,B 0,C 180,E1 8670.423,E2 8670.423} C_VEL
LIN {X 0,Y 262.461,Z 1047.011,A -85,B 0,C 180,E1 8667.42,E2 8667.42} C_VEL
LIN {X 0,Y 275.022,Z 1031.681,A -85,B 0,C 180,E1 8665.138,E2 8665.138} C_VEL
LIN {X 0,Y 289.075,Z 1012.552,A -85,B 0,C 180,E1 8662.889,E2 8662.889} C_VEL
LIN {X 0,Y 300.82,Z 994.633,A -85,B 0,C 180,E1 8661.221,E2 8661.221} C_VEL
LIN {X 0,Y 312.328,Z 974.659,A -85,B 0,C 180,E1 8659.742,E2 8659.742} C_VEL
LIN {X 0,Y 322.248,Z 955.031,A -85,B 0,C 180,E1 8658.571,E2 8658.571} C_VEL
LIN {X 0,Y 331.815,Z 932.84,A -85,B 0,C 180,E1 8657.523,E2 8657.523} C_VEL
LIN {X 0,Y 339.365,Z 912.181,A -85,B 0,C 180,E1 8656.75,E2 8656.75} C_VEL
LIN {X 0,Y 346.282,Z 888.782,A -85,B 0,C 180,E1 8656.073,E2 8656.073} C_VEL
LIN {X 0,Y 351.481,Z 866.456,A -85,B 0,C 180,E1 8655.585,E2 8655.585} C_VEL
LIN {X 0,Y 355.411,Z 842.166,A -85,B 0,C 180,E1 8655.174,E2 8655.174} C_VEL
LIN {X 0,Y 370.892,Z 695.586,A -85,B 0,C 180,E1 8653.069,E2 8653.069} C_VEL
LIN {X 0,Y 368.931,Z 689.932,A -85,B 0,C 180,E1 8650.778,E2 8650.778} C_VEL
LIN {X 0,Y 367.277,Z 685.115,A -85,B 0,C 180,E1 8648.217,E2 8648.217} C_VEL
LIN {X 0,Y 366.093,Z 681.44,A -85,B 0,C 180,E1 8645.328,E2 8645.328} C_VEL
LIN {X 0,Y 365.608,Z 679.379,A -85,B 0,C 180,E1 8641.097,E2 8641.097} C_VEL
LIN {X 0,Y 365.996,Z 679.944,A -85,B 0,C 180,E1 8638.748,E2 8638.748} C_VEL
LIN {X 0,Y 367.491,Z 682.864,A -85,B 0,C 180,E1 8635.24,E2 8635.24} C_VEL
LIN {X 0,Y 369.304,Z 686.886,A -85,B 0,C 180,E1 8632.611,E2 8632.611} C_VEL
LIN {X 0,Y 371.556,Z 692.01,A -85,B 0,C 180,E1 8630.142,E2 8630.142} C_VEL
LIN {X 0,Y 363.586,Z 766.389,A -85,B 0,C 180,E1 8629.073,E2 8629.073} C_VEL
LIN {X 0,Y 362.56,Z 774.081,A -85,B 0,C 180,E1 8629.109,E2 8629.109} C_VEL
LIN {X 0,Y 359.045,Z 794.605,A -85,B 0,C 180,E1 8629.789,E2 8629.789} C_VEL
LIN {X 0,Y 358.183,Z 801.208,A -85,B 0,C 180,E1 8629.811,E2 8629.811} C_VEL
LIN {X 0,Y 352.747,Z 848.47,A -85,B 0,C 180,E1 8629.116,E2 8629.116} C_VEL
LIN {X 0,Y 348.203,Z 872.349,A -85,B 0,C 180,E1 8628.683,E2 8628.683} C_VEL
LIN {X 0,Y 342.274,Z 895.904,A -85,B 0,C 180,E1 8628.138,E2 8628.138} C_VEL
LIN {X 0,Y 334.976,Z 918.42,A -85,B 0,C 180,E1 8627.445,E2 8627.445} C_VEL
LIN {X 0,Y 326.385,Z 940.628,A -85,B 0,C 180,E1 8626.575,E2 8626.575} C_VEL
LIN {X 0,Y 316.974,Z 961.028,A -85,B 0,C 180,E1 8625.565,E2 8625.565} C_VEL
LIN {X 0,Y 305.871,Z 982.105,A -85,B 0,C 180,E1 8624.272,E2 8624.272} C_VEL
LIN {X 0,Y 294.14,Z 1001.349,A -85,B 0,C 180,E1 8622.79,E2 8622.79} C_VEL
LIN {X 0,Y 281.342,Z 1020.227,A -85,B 0,C 180,E1 8620.974,E2 8620.974} C_VEL
LIN {X 0,Y 268.012,Z 1037.603,A -85,B 0,C 180,E1 8618.859,E2 8618.859} C_VEL
LIN {X 0,Y 253.513,Z 1054.825,A -85,B 0,C 180,E1 8616.212,E2 8616.212} C_VEL
LIN {X 0,Y 239.601,Z 1069.714,A -85,B 0,C 180,E1 8613.26,E2 8613.26} C_VEL
LIN {X 0,Y 224.925,Z 1084.276,A -85,B 0,C 180,E1 8609.55,E2 8609.55} C_VEL
LIN {X 0,Y 211.386,Z 1096.643,A -85,B 0,C 180,E1 8605.391,E2 8605.391} C_VEL
LIN {X 0,Y 197.838,Z 1108.406,A -85,B 0,C 180,E1 8600.195,E2 8600.195} C_VEL
LIN {X 0,Y 186.536,Z 1117.788,A -85,B 0,C 180,E1 8594.604,E2 8594.604} C_VEL
LIN {X 0,Y 175.871,Z 1126.659,A -85,B 0,C 180,E1 8587.469,E2 8587.469} C_VEL
LIN {X 0,Y 168.738,Z 1132.788,A -85,B 0,C 180,E1 8580.638,E2 8580.638} C_VEL
LIN {X 0,Y 163.329,Z 1138.135,A -85,B 0,C 180,E1 8572.42,E2 8572.42} C_VEL
LIN {X 0,Y 160.755,Z 1141.364,A -85,B 0,C 180,E1 8564.775,E2 8564.775} C_VEL
LIN {X 0,Y 160.015,Z 1143.089,A -85,B 0,C 180,E1 8558.263,E2 8558.263} C_VEL
LIN {X 0,Y 160.004,Z 1143.812,A -85,B 0,C 180,E1 8552.507,E2 8552.507} C_VEL
LIN {X 0,Y 160.004,Z 1143.806,A -85,B 0,C 180,E1 8547.493,E2 8547.493} C_VEL
LIN {X 0,Y 160.016,Z 1143.072,A -85,B 0,C 180,E1 8541.737,E2 8541.737} C_VEL
LIN {X 0,Y 160.755,Z 1141.334,A -85,B 0,C 180,E1 8535.225,E2 8535.225} C_VEL
LIN {X 0,Y 163.622,Z 1137.782,A -85,B 0,C 180,E1 8526.977,E2 8526.977} C_VEL
LIN {X 0,Y 169.022,Z 1132.46,A -85,B 0,C 180,E1 8519.024,E2 8519.024} C_VEL
LIN {X 0,Y 177.055,Z 1125.628,A -85,B 0,C 180,E1 8511.595,E2 8511.595} C_VEL
LIN {X 0,Y 187.528,Z 1116.85,A -85,B 0,C 180,E1 8504.834,E2 8504.834} C_VEL
LIN {X 0,Y 199.58,Z 1106.823,A -85,B 0,C 180,E1 8499.054,E2 8499.054} C_VEL
LIN {X 0,Y 212.679,Z 1095.321,A -85,B 0,C 180,E1 8494.162,E2 8494.162} C_VEL
LIN {X 0,Y 227.149,Z 1081.948,A -85,B 0,C 180,E1 8489.829,E2 8489.829} C_VEL
LIN {X 0,Y 240.34,Z 1068.714,A -85,B 0,C 180,E1 8486.559,E2 8486.559} C_VEL
LIN {X 0,Y 255.081,Z 1052.79,A -85,B 0,C 180,E1 8483.471,E2 8483.471} C_VEL
LIN {X 0,Y 268.818,Z 1036.281,A -85,B 0,C 180,E1 8480.994,E2 8480.994} C_VEL
LIN {X 0,Y 282.592,Z 1018.096,A -85,B 0,C 180,E1 8478.827,E2 8478.827} C_VEL
LIN {X 0,Y 294.986,Z 999.596,A -85,B 0,C 180,E1 8477.084,E2 8477.084} C_VEL
LIN {X 0,Y 307.215,Z 979.179,A -85,B 0,C 180,E1 8475.55,E2 8475.55} C_VEL
LIN {X 0,Y 317.402,Z 959.576,A -85,B 0,C 180,E1 8474.372,E2 8474.372} C_VEL
LIN {X 0,Y 327.271,Z 937.838,A -85,B 0,C 180,E1 8473.32,E2 8473.32} C_VEL
LIN {X 0,Y 335.417,Z 916.341,A -85,B 0,C 180,E1 8472.5,E2 8472.5} C_VEL
LIN {X 0,Y 342.866,Z 892.728,A -85,B 0,C 180,E1 8471.794,E2 8471.794} C_VEL
LIN {X 0,Y 348.387,Z 870.155,A -85,B 0,C 180,E1 8471.285,E2 8471.285} C_VEL
LIN {X 0,Y 352.89,Z 845.122,A -85,B 0,C 180,E1 8470.844,E2 8470.844} C_VEL
LIN {X 0,Y 365.43,Z 731.483,A -85,B 0,C 180,E1 8469.202,E2 8469.202} C_VEL
LIN {X 0,Y 369.129,Z 697.545,A -85,B 0,C 180,E1 8468.725,E2 8468.725} C_VEL
LIN {X 0,Y 367.037,Z 692.599,A -85,B 0,C 180,E1 8466.099,E2 8466.099} C_VEL
LIN {X 0,Y 365.761,Z 689.697,A -85,B 0,C 180,E1 8463.919,E2 8463.919} C_VEL
LIN {X 0,Y 364.525,Z 687.061,A -85,B 0,C 180,E1 8460.314,E2 8460.314} C_VEL
LIN {X 0,Y 364.28,Z 687.101,A -85,B 0,C 180,E1 8458.112,E2 8458.112} C_VEL
LIN {X 0,Y 364.925,Z 689.735,A -85,B 0,C 180,E1 8454.055,E2 8454.055} C_VEL
LIN {X 0,Y 366.267,Z 693.943,A -85,B 0,C 180,E1 8451.127,E2 8451.127} C_VEL
LIN {X 0,Y 368.181,Z 699.669,A -85,B 0,C 180,E1 8448.406,E2 8448.406} C_VEL
LIN {X 0,Y 368.523,Z 701.054,A -85,B 0,C 180,E1 8447.959,E2 8447.959} C_VEL
LIN {X 0,Y 352.869,Z 845.594,A -85,B 0,C 180,E1 8445.937,E2 8445.937} C_VEL
LIN {X 0,Y 348.451,Z 870.432,A -85,B 0,C 180,E1 8445.513,E2 8445.513} C_VEL
LIN {X 0,Y 342.967,Z 892.936,A -85,B 0,C 180,E1 8445.019,E2 8445.019} C_VEL
LIN {X 0,Y 335.909,Z 915.405,A -85,B 0,C 180,E1 8444.357,E2 8444.357} C_VEL
LIN {X 0,Y 328.317,Z 935.563,A -85,B 0,C 180,E1 8443.605,E2 8443.605} C_VEL
LIN {X 0,Y 318.577,Z 957.292,A -85,B 0,C 180,E1 8442.582,E2 8442.582} C_VEL
LIN {X 0,Y 308.952,Z 975.884,A -85,B 0,C 180,E1 8441.49,E2 8441.49} C_VEL
LIN {X 0,Y 296.448,Z 996.909,A -85,B 0,C 180,E1 8439.944,E2 8439.944} C_VEL
LIN {X 0,Y 284.611,Z 1014.503,A -85,B 0,C 180,E1 8438.317,E2 8438.317} C_VEL
LIN {X 0,Y 270.617,Z 1032.939,A -85,B 0,C 180,E1 8436.154,E2 8436.154} C_VEL
LIN {X 0,Y 257.377,Z 1048.667,A -85,B 0,C 180,E1 8433.821,E2 8433.821} C_VEL
LIN {X 0,Y 242.748,Z 1064.271,A -85,B 0,C 180,E1 8430.838,E2 8430.838} C_VEL
LIN {X 0,Y 228.86,Z 1077.895,A -85,B 0,C 180,E1 8427.482,E2 8427.482} C_VEL
LIN {X 0,Y 215.051,Z 1090.213,A -85,B 0,C 180,E1 8423.477,E2 8423.477} C_VEL
LIN {X 0,Y 202.003,Z 1101.2,A -85,B 0,C 180,E1 8418.797,E2 8418.797} C_VEL
LIN {X 0,Y 189.79,Z 1110.776,A -85,B 0,C 180,E1 8413.227,E2 8413.227} C_VEL
LIN {X 0,Y 179.477,Z 1118.759,A -85,B 0,C 180,E1 8406.991,E2 8406.991} C_VEL
LIN {X 0,Y 170.96,Z 1125.208,A -85,B 0,C 180,E1 8399.811,E2 8399.811} C_VEL
LIN {X 0,Y 164.883,Z 1130.241,A -85,B 0,C 180,E1 8391.9,E2 8391.9} C_VEL
LIN {X 0,Y 161.513,Z 1133.362,A -85,B 0,C 180,E1 8383.972,E2 8383.972} C_VEL
LIN {X 0,Y 160.264,Z 1135.009,A -85,B 0,C 180,E1 8376.808,E2 8376.808} C_VEL
LIN {X 0,Y 160.048,Z 1135.563,A -85,B 0,C 180,E1 8369.642,E2 8369.642} C_VEL
LIN {X 0,Y 160.327,Z 1134.913,A -85,B 0,C 180,E1 8362.474,E2 8362.474} C_VEL
LIN {X 0,Y 161.588,Z 1133.31,A -85,B 0,C 180,E1 8355.669,E2 8355.669} C_VEL
LIN {X 0,Y 165.143,Z 1130.068,A -85,B 0,C 180,E1 8347.577,E2 8347.577} C_VEL
LIN {X 0,Y 171.305,Z 1125.013,A -85,B 0,C 180,E1 8339.754,E2 8339.754} C_VEL
LIN {X 0,Y 180.239,Z 1118.242,A -85,B 0,C 180,E1 8332.393,E2 8332.393} C_VEL
LIN {X 0,Y 190.205,Z 1110.575,A -85,B 0,C 180,E1 8326.476,E2 8326.476} C_VEL
LIN {X 0,Y 202.485,Z 1100.936,A -85,B 0,C 180,E1 8320.928,E2 8320.928} C_VEL
LIN {X 0,Y 215.702,Z 1089.825,A -85,B 0,C 180,E1 8316.237,E2 8316.237} C_VEL
LIN {X 0,Y 230.16,Z 1076.842,A -85,B 0,C 180,E1 8312.097,E2 8312.097} C_VEL
LIN {X 0,Y 243.377,Z 1063.873,A -85,B 0,C 180,E1 8308.944,E2 8308.944} C_VEL
LIN {X 0,Y 258.121,Z 1048.088,A -85,B 0,C 180,E1 8305.959,E2 8305.959} C_VEL
LIN {X 0,Y 271.236,Z 1032.495,A -85,B 0,C 180,E1 8303.667,E2 8303.667} C_VEL
LIN {X 0,Y 285.748,Z 1013.253,A -85,B 0,C 180,E1 8301.441,E2 8301.441} C_VEL
LIN {X 0,Y 297.48,Z 995.744,A -85,B 0,C 180,E1 8299.845,E2 8299.845} C_VEL
LIN {X 0,Y 309.708,Z 975.012,A -85,B 0,C 180,E1 8298.344,E2 8298.344} C_VEL
LIN {X 0,Y 319.345,Z 956.31,A -85,B 0,C 180,E1 8297.257,E2 8297.257} C_VEL
LIN {X 0,Y 329.496,Z 933.311,A -85,B 0,C 180,E1 8296.197,E2 8296.197} C_VEL
LIN {X 0,Y 336.829,Z 913.629,A -85,B 0,C 180,E1 8295.481,E2 8295.481} C_VEL
LIN {X 0,Y 344.193,Z 889.385,A -85,B 0,C 180,E1 8294.795,E2 8294.795} C_VEL
LIN {X 0,Y 349.369,Z 867.596,A -85,B 0,C 180,E1 8294.332,E2 8294.332} C_VEL
LIN {X 0,Y 353.518,Z 842.873,A -85,B 0,C 180,E1 8293.922,E2 8293.922} C_VEL
LIN {X 0,Y 368.821,Z 701.064,A -85,B 0,C 180,E1 8291.936,E2 8291.936} C_VEL
LIN {X 0,Y 367.309,Z 696.571,A -85,B 0,C 180,E1 8289.954,E2 8289.954} C_VEL
LIN {X 0,Y 366.015,Z 692.423,A -85,B 0,C 180,E1 8287.693,E2 8287.693} C_VEL
LIN {X 0,Y 365.026,Z 689.235,A -85,B 0,C 180,E1 8285.029,E2 8285.029} C_VEL
LIN {X 0,Y 364.644,Z 687.309,A -85,B 0,C 180,E1 8280.943,E2 8280.943} C_VEL
LIN {X 0,Y 365.048,Z 688.04,A -85,B 0,C 180,E1 8278.587,E2 8278.587} C_VEL
LIN {X 0,Y 366.404,Z 690.775,A -85,B 0,C 180,E1 8275.382,E2 8275.382} C_VEL
LIN {X 0,Y 368.109,Z 694.709,A -85,B 0,C 180,E1 8272.822,E2 8272.822} C_VEL
LIN {X 0,Y 369.389,Z 697.897,A -85,B 0,C 180,E1 8271.276,E2 8271.276} C_VEL
LIN {X 0,Y 358.183,Z 801.208,A -85,B 0,C 180,E1 8269.811,E2 8269.811} C_VEL
LIN {X 0,Y 357.174,Z 808.904,A -85,B 0,C 180,E1 8269.856,E2 8269.856} C_VEL
LIN {X 0,Y 353.723,Z 829.418,A -85,B 0,C 180,E1 8270.561,E2 8270.561} C_VEL
LIN {X 0,Y 352.758,Z 836.004,A -85,B 0,C 180,E1 8270.581,E2 8270.581} C_VEL
LIN {X 0,Y 349.347,Z 858.462,A -85,B 0,C 180,E1 8270.226,E2 8270.226} C_VEL
LIN {X 0,Y 343.668,Z 884.254,A -85,B 0,C 180,E1 8269.721,E2 8269.721} C_VEL
LIN {X 0,Y 337.696,Z 904.959,A -85,B 0,C 180,E1 8269.201,E2 8269.201} C_VEL
LIN {X 0,Y 329.169,Z 928.933,A -85,B 0,C 180,E1 8268.418,E2 8268.418} C_VEL
LIN {X 0,Y 320.486,Z 949.311,A -85,B 0,C 180,E1 8267.565,E2 8267.565} C_VEL
LIN {X 0,Y 309.137,Z 972.028,A -85,B 0,C 180,E1 8266.36,E2 8266.36} C_VEL
LIN {X 0,Y 298.46,Z 990.596,A -85,B 0,C 180,E1 8265.134,E2 8265.134} C_VEL
LIN {X 0,Y 284.837,Z 1011.398,A -85,B 0,C 180,E1 8263.404,E2 8263.404} C_VEL
LIN {X 0,Y 272.313,Z 1028.422,A -85,B 0,C 180,E1 8261.621,E2 8261.621} C_VEL
LIN {X 0,Y 257.669,Z 1046.232,A -85,B 0,C 180,E1 8259.262,E2 8259.262} C_VEL
LIN {X 0,Y 244.669,Z 1060.575,A -85,B 0,C 180,E1 8256.855,E2 8256.855} C_VEL
LIN {X 0,Y 228.339,Z 1076.974,A -85,B 0,C 180,E1 8253.293,E2 8253.293} C_VEL
LIN {X 0,Y 214.414,Z 1089.807,A -85,B 0,C 180,E1 8249.624,E2 8249.624} C_VEL
LIN {X 0,Y 199.507,Z 1102.526,A -85,B 0,C 180,E1 8244.779,E2 8244.779} C_VEL
LIN {X 0,Y 187.318,Z 1112.406,A -85,B 0,C 180,E1 8239.758,E2 8239.758} C_VEL
LIN {X 0,Y 175.191,Z 1121.874,A -85,B 0,C 180,E1 8233.228,E2 8233.228} C_VEL
LIN {X 0,Y 166.182,Z 1128.94,A -85,B 0,C 180,E1 8226.56,E2 8226.56} C_VEL
LIN {X 0,Y 158.309,Z 1135.486,A -85,B 0,C 180,E1 8217.84,E2 8217.84} C_VEL
LIN {X 0,Y 154.237,Z 1139.472,A -85,B 0,C 180,E1 8210.096,E2 8210.096} C_VEL
LIN {X 0,Y 152.234,Z 1142.37,A -85,B 0,C 180,E1 8201.364,E2 8201.364} C_VEL
LIN {X 0,Y 151.986,Z 1143.479,A -85,B 0,C 180,E1 8194.528,E2 8194.528} C_VEL
LIN {X 0,Y 152.027,Z 1143.678,A -85,B 0,C 180,E1 8188.643,E2 8188.643} C_VEL
LIN {X 0,Y 152.002,Z 1143.077,A -85,B 0,C 180,E1 8182.44,E2 8182.44} C_VEL
LIN {X 0,Y 152.737,Z 1141.359,A -85,B 0,C 180,E1 8175.208,E2 8175.208} C_VEL
LIN {X 0,Y 155.179,Z 1138.429,A -85,B 0,C 180,E1 8167.656,E2 8167.656} C_VEL
LIN {X 0,Y 161.072,Z 1133.031,A -85,B 0,C 180,E1 8158.57,E2 8158.57} C_VEL
LIN {X 0,Y 168.537,Z 1126.984,A -85,B 0,C 180,E1 8151.469,E2 8151.469} C_VEL
LIN {X 0,Y 179.832,Z 1118.156,A -85,B 0,C 180,E1 8144.029,E2 8144.029} C_VEL
LIN {X 0,Y 191.41,Z 1109,A -85,B 0,C 180,E1 8138.411,E2 8138.411} C_VEL
LIN {X 0,Y 206.219,Z 1096.737,A -85,B 0,C 180,E1 8132.892,E2 8132.892} C_VEL
LIN {X 0,Y 219.425,Z 1085.107,A -85,B 0,C 180,E1 8128.964,E2 8128.964} C_VEL
LIN {X 0,Y 235.206,Z 1070.029,A -85,B 0,C 180,E1 8125.11,E2 8125.11} C_VEL
LIN {X 0,Y 248.664,Z 1056.042,A -85,B 0,C 180,E1 8122.355,E2 8122.355} C_VEL
LIN {X 0,Y 263.528,Z 1039.009,A -85,B 0,C 180,E1 8119.736,E2 8119.736} C_VEL
LIN {X 0,Y 276.608,Z 1022.42,A -85,B 0,C 180,E1 8117.728,E2 8117.728} C_VEL
LIN {X 0,Y 290.491,Z 1002.648,A -85,B 0,C 180,E1 8115.833,E2 8115.833} C_VEL
LIN {X 0,Y 302.002,Z 984.206,A -85,B 0,C 180,E1 8114.434,E2 8114.434} C_VEL
LIN {X 0,Y 313.673,Z 962.805,A -85,B 0,C 180,E1 8113.134,E2 8113.134} C_VEL
LIN {X 0,Y 322.752,Z 943.628,A -85,B 0,C 180,E1 8112.197,E2 8112.197} C_VEL
LIN {X 0,Y 332.372,Z 919.664,A -85,B 0,C 180,E1 8111.267,E2 8111.267} C_VEL
LIN {X 0,Y 339.529,Z 898.074,A -85,B 0,C 180,E1 8110.618,E2 8110.618} C_VEL
LIN {X 0,Y 345.967,Z 873.434,A -85,B 0,C 180,E1 8110.056,E2 8110.056} C_VEL
LIN {X 0,Y 350.426,Z 850.619,A -85,B 0,C 180,E1 8109.653,E2 8109.653} C_VEL
LIN {X 0,Y 354.805,Z 815.146,A -85,B 0,C 180,E1 8109.132,E2 8109.132} C_VEL
LIN {X 0,Y 367.091,Z 703.315,A -85,B 0,C 180,E1 8107.552,E2 8107.552} C_VEL
LIN {X 0,Y 365.48,Z 699.519,A -85,B 0,C 180,E1 8105.259,E2 8105.259} C_VEL
LIN {X 0,Y 364.614,Z 697.45,A -85,B 0,C 180,E1 8103.616,E2 8103.616} C_VEL
LIN {X 0,Y 363.521,Z 694.956,A -85,B 0,C 180,E1 8100.158,E2 8100.158} C_VEL
LIN {X 0,Y 363.297,Z 695.138,A -85,B 0,C 180,E1 8097.95,E2 8097.95} C_VEL
LIN {X 0,Y 363.873,Z 697.588,A -85,B 0,C 180,E1 8094.244,E2 8094.244} C_VEL
LIN {X 0,Y 365.158,Z 701.818,A -85,B 0,C 180,E1 8091.306,E2 8091.306} C_VEL
LIN {X 0,Y 366.576,Z 706.463,A -85,B 0,C 180,E1 8089.116,E2 8089.116} C_VEL
LIN {X 0,Y 351.235,Z 845.515,A -85,B 0,C 180,E1 8087.215,E2 8087.215} C_VEL
LIN {X 0,Y 346.746,Z 870.427,A -85,B 0,C 180,E1 8086.804,E2 8086.804} C_VEL
LIN {X 0,Y 341.222,Z 892.817,A -85,B 0,C 180,E1 8086.332,E2 8086.332} C_VEL
LIN {X 0,Y 333.845,Z 915.956,A -85,B 0,C 180,E1 8085.676,E2 8085.676} C_VEL
LIN {X 0,Y 325.701,Z 937.172,A -85,B 0,C 180,E1 8084.908,E2 8084.908} C_VEL
LIN {X 0,Y 315.822,Z 958.586,A -85,B 0,C 180,E1 8083.92,E2 8083.92} C_VEL
LIN {X 0,Y 305.043,Z 978.91,A -85,B 0,C 180,E1 8082.746,E2 8082.746} C_VEL
LIN {X 0,Y 292.917,Z 998.547,A -85,B 0,C 180,E1 8081.31,E2 8081.31} C_VEL
LIN {X 0,Y 280.033,Z 1017.195,A -85,B 0,C 180,E1 8079.602,E2 8079.602} C_VEL
LIN {X 0,Y 266.171,Z 1034.757,A -85,B 0,C 180,E1 8077.536,E2 8077.536} C_VEL
LIN {X 0,Y 251.495,Z 1051.557,A -85,B 0,C 180,E1 8075.024,E2 8075.024} C_VEL
LIN {X 0,Y 237.355,Z 1066.036,A -85,B 0,C 180,E1 8072.21,E2 8072.21} C_VEL
LIN {X 0,Y 222.4,Z 1080.07,A -85,B 0,C 180,E1 8068.675,E2 8068.675} C_VEL
LIN {X 0,Y 209.052,Z 1091.477,A -85,B 0,C 180,E1 8064.875,E2 8064.875} C_VEL
LIN {X 0,Y 194.877,Z 1102.82,A -85,B 0,C 180,E1 8059.863,E2 8059.863} C_VEL
LIN {X 0,Y 182.851,Z 1111.789,A -85,B 0,C 180,E1 8054.423,E2 8054.423} C_VEL
LIN {X 0,Y 171.263,Z 1120.179,A -85,B 0,C 180,E1 8047.387,E2 8047.387} C_VEL
LIN {X 0,Y 162.946,Z 1126.166,A -85,B 0,C 180,E1 8040.211,E2 8040.211} C_VEL
LIN {X 0,Y 156.43,Z 1131.147,A -85,B 0,C 180,E1 8031.367,E2 8031.367} C_VEL
LIN {X 0,Y 153.375,Z 1133.901,A -85,B 0,C 180,E1 8023.574,E2 8023.574} C_VEL
LIN {X 0,Y 152.16,Z 1135.484,A -85,B 0,C 180,E1 8015.279,E2 8015.279} C_VEL
LIN {X 0,Y 152.053,Z 1135.707,A -85,B 0,C 180,E1 8008.493,E2 8008.493} C_VEL
LIN {X 0,Y 152.406,Z 1135.059,A -85,B 0,C 180,E1 8001.701,E2 8001.701} C_VEL
LIN {X 0,Y 153.881,Z 1133.414,A -85,B 0,C 180,E1 7994.549,E2 7994.549} C_VEL
LIN {X 0,Y 158.12,Z 1129.882,A -85,B 0,C 180,E1 7985.73,E2 7985.73} C_VEL
LIN {X 0,Y 164.553,Z 1125.054,A -85,B 0,C 180,E1 7978.086,E2 7978.086} C_VEL
LIN {X 0,Y 174.298,Z 1118.114,A -85,B 0,C 180,E1 7970.448,E2 7970.448} C_VEL
LIN {X 0,Y 184.914,Z 1110.396,A -85,B 0,C 180,E1 7964.458,E2 7964.458} C_VEL
LIN {X 0,Y 198.5,Z 1100.131,A -85,B 0,C 180,E1 7958.654,E2 7958.654} C_VEL
LIN {X 0,Y 211.674,Z 1089.486,A -85,B 0,C 180,E1 7954.243,E2 7954.243} C_VEL
LIN {X 0,Y 227.414,Z 1075.695,A -85,B 0,C 180,E1 7949.983,E2 7949.983} C_VEL
LIN {X 0,Y 241.632,Z 1062.072,A -85,B 0,C 180,E1 7946.811,E2 7946.811} C_VEL
LIN {X 0,Y 256.213,Z 1046.603,A -85,B 0,C 180,E1 7944.047,E2 7944.047} C_VEL
LIN {X 0,Y 270.222,Z 1030.199,A -85,B 0,C 180,E1 7941.756,E2 7941.756} C_VEL
LIN {X 0,Y 283.754,Z 1012.337,A -85,B 0,C 180,E1 7939.804,E2 7939.804} C_VEL
LIN {X 0,Y 295.855,Z 994.517,A -85,B 0,C 180,E1 7938.251,E2 7938.251} C_VEL
LIN {X 0,Y 307.717,Z 974.56,A -85,B 0,C 180,E1 7936.873,E2 7936.873} C_VEL
LIN {X 0,Y 317.954,Z 954.906,A -85,B 0,C 180,E1 7935.782,E2 7935.782} C_VEL
LIN {X 0,Y 327.851,Z 932.546,A -85,B 0,C 180,E1 7934.805,E2 7934.805} C_VEL
LIN {X 0,Y 335.569,Z 911.972,A -85,B 0,C 180,E1 7934.095,E2 7934.095} C_VEL
LIN {X 0,Y 342.614,Z 888.716,A -85,B 0,C 180,E1 7933.474,E2 7933.474} C_VEL
LIN {X 0,Y 347.916,Z 866.529,A -85,B 0,C 180,E1 7933.025,E2 7933.025} C_VEL
LIN {X 0,Y 351.968,Z 842.261,A -85,B 0,C 180,E1 7932.638,E2 7932.638} C_VEL
LIN {X 0,Y 366.872,Z 706.545,A -85,B 0,C 180,E1 7930.768,E2 7930.768} C_VEL
LIN {X 0,Y 365.061,Z 700.765,A -85,B 0,C 180,E1 7927.792,E2 7927.792} C_VEL
LIN {X 0,Y 364.013,Z 697.122,A -85,B 0,C 180,E1 7924.885,E2 7924.885} C_VEL
LIN {X 0,Y 363.669,Z 695.25,A -85,B 0,C 180,E1 7920.945,E2 7920.945} C_VEL
LIN {X 0,Y 364.02,Z 695.915,A -85,B 0,C 180,E1 7918.741,E2 7918.741} C_VEL
LIN {X 0,Y 365.279,Z 698.572,A -85,B 0,C 180,E1 7915.604,E2 7915.604} C_VEL
LIN {X 0,Y 366.919,Z 702.531,A -85,B 0,C 180,E1 7913.035,E2 7913.035} C_VEL
LIN {X 0,Y 367.374,Z 703.852,A -85,B 0,C 180,E1 7912.423,E2 7912.423} C_VEL
LIN {X 0,Y 352.758,Z 836.004,A -85,B 0,C 180,E1 7910.581,E2 7910.581} C_VEL
LIN {X 0,Y 351.564,Z 843.667,A -85,B 0,C 180,E1 7910.63,E2 7910.63} C_VEL
LIN {X 0,Y 346.992,Z 863.991,A -85,B 0,C 180,E1 7911.319,E2 7911.319} C_VEL
LIN {X 0,Y 345.419,Z 870.476,A -85,B 0,C 180,E1 7911.315,E2 7911.315} C_VEL
LIN {X 0,Y 339.675,Z 893.327,A -85,B 0,C 180,E1 7910.84,E2 7910.84} C_VEL
LIN {X 0,Y 332.262,Z 916.155,A -85,B 0,C 180,E1 7910.211,E2 7910.211} C_VEL
LIN {X 0,Y 324.391,Z 936.428,A -85,B 0,C 180,E1 7909.507,E2 7909.507} C_VEL
LIN {X 0,Y 314.23,Z 958.431,A -85,B 0,C 180,E1 7908.542,E2 7908.542} C_VEL
LIN {X 0,Y 304.172,Z 977.318,A -85,B 0,C 180,E1 7907.506,E2 7907.506} C_VEL
LIN {X 0,Y 291.067,Z 998.702,A -85,B 0,C 180,E1 7906.04,E2 7906.04} C_VEL
LIN {X 0,Y 278.629,Z 1016.636,A -85,B 0,C 180,E1 7904.482,E2 7904.482} C_VEL
LIN {X 0,Y 263.821,Z 1035.526,A -85,B 0,C 180,E1 7902.402,E2 7902.402} C_VEL
LIN {X 0,Y 249.825,Z 1051.598,A -85,B 0,C 180,E1 7900.146,E2 7900.146} C_VEL
LIN {X 0,Y 234.235,Z 1067.665,A -85,B 0,C 180,E1 7897.228,E2 7897.228} C_VEL
LIN {X 0,Y 220.103,Z 1081.006,A -85,B 0,C 180,E1 7894.091,E2 7894.091} C_VEL
LIN {X 0,Y 204.544,Z 1094.431,A -85,B 0,C 180,E1 7889.911,E2 7889.911} C_VEL
LIN {X 0,Y 190.866,Z 1105.451,A -85,B 0,C 180,E1 7885.334,E2 7885.334} C_VEL
LIN {X 0,Y 176.788,Z 1116.099,A -85,B 0,C 180,E1 7879.279,E2 7879.279} C_VEL
LIN {X 0,Y 165.801,Z 1124.193,A -85,B 0,C 180,E1 7872.958,E2 7872.958} C_VEL
LIN {X 0,Y 155.66,Z 1131.668,A -85,B 0,C 180,E1 7864.693,E2 7864.693} C_VEL
LIN {X 0,Y 149.313,Z 1136.759,A -85,B 0,C 180,E1 7856.659,E2 7856.659} C_VEL
LIN {X 0,Y 145.272,Z 1140.697,A -85,B 0,C 180,E1 7847.215,E2 7847.215} C_VEL
LIN {X 0,Y 144.09,Z 1142.594,A -85,B 0,C 180,E1 7839.587,E2 7839.587} C_VEL
LIN {X 0,Y 143.998,Z 1143.343,A -85,B 0,C 180,E1 7833.583,E2 7833.583} C_VEL
LIN {X 0,Y 144.017,Z 1143.434,A -85,B 0,C 180,E1 7828.011,E2 7828.011} C_VEL
LIN {X 0,Y 144.022,Z 1142.793,A -85,B 0,C 180,E1 7821.617,E2 7821.617} C_VEL
LIN {X 0,Y 144.973,Z 1141.026,A -85,B 0,C 180,E1 7813.985,E2 7813.985} C_VEL
LIN {X 0,Y 148.216,Z 1137.713,A -85,B 0,C 180,E1 7805.275,E2 7805.275} C_VEL
LIN {X 0,Y 154.414,Z 1132.548,A -85,B 0,C 180,E1 7796.605,E2 7796.605} C_VEL
LIN {X 0,Y 163.047,Z 1126.122,A -85,B 0,C 180,E1 7788.964,E2 7788.964} C_VEL
LIN {X 0,Y 174.541,Z 1117.646,A -85,B 0,C 180,E1 7781.864,E2 7781.864} C_VEL
LIN {X 0,Y 186.997,Z 1108.305,A -85,B 0,C 180,E1 7776.156,E2 7776.156} C_VEL
LIN {X 0,Y 201.705,Z 1096.608,A -85,B 0,C 180,E1 7770.952,E2 7770.952} C_VEL
LIN {X 0,Y 215.533,Z 1084.871,A -85,B 0,C 180,E1 7767.036,E2 7767.036} C_VEL
LIN {X 0,Y 231.023,Z 1070.562,A -85,B 0,C 180,E1 7763.428,E2 7763.428} C_VEL
LIN {X 0,Y 244.818,Z 1056.645,A -85,B 0,C 180,E1 7760.725,E2 7760.725} C_VEL
LIN {X 0,Y 260.802,Z 1038.81,A -85,B 0,C 180,E1 7758.045,E2 7758.045} C_VEL
LIN {X 0,Y 273.783,Z 1022.694,A -85,B 0,C 180,E1 7756.155,E2 7756.155} C_VEL
LIN {X 0,Y 287.92,Z 1003.001,A -85,B 0,C 180,E1 7754.323,E2 7754.323} C_VEL
LIN {X 0,Y 299.619,Z 984.605,A -85,B 0,C 180,E1 7752.975,E2 7752.975} C_VEL
LIN {X 0,Y 311.969,Z 962.312,A -85,B 0,C 180,E1 7751.672,E2 7751.672} C_VEL
LIN {X 0,Y 321.181,Z 943.085,A -85,B 0,C 180,E1 7750.776,E2 7750.776} C_VEL
LIN {X 0,Y 330.648,Z 919.765,A -85,B 0,C 180,E1 7749.913,E2 7749.913} C_VEL
LIN {X 0,Y 337.714,Z 898.756,A -85,B 0,C 180,E1 7749.305,E2 7749.305} C_VEL
LIN {X 0,Y 344.383,Z 873.698,A -85,B 0,C 180,E1 7748.754,E2 7748.754} C_VEL
LIN {X 0,Y 348.867,Z 851.098,A -85,B 0,C 180,E1 7748.37,E2 7748.37} C_VEL
LIN {X 0,Y 353.161,Z 817.189,A -85,B 0,C 180,E1 7747.884,E2 7747.884} C_VEL
LIN {X 0,Y 365.208,Z 709.441,A -85,B 0,C 180,E1 7746.406,E2 7746.406} C_VEL
LIN {X 0,Y 363.627,Z 705.444,A -85,B 0,C 180,E1 7743.626,E2 7743.626} C_VEL
LIN {X 0,Y 362.518,Z 702.857,A -85,B 0,C 180,E1 7740,E2 7740} C_VEL
LIN {X 0,Y 362.319,Z 703.107,A -85,B 0,C 180,E1 7737.944,E2 7737.944} C_VEL
LIN {X 0,Y 362.817,Z 705.397,A -85,B 0,C 180,E1 7734.465,E2 7734.465} C_VEL
LIN {X 0,Y 363.974,Z 709.463,A -85,B 0,C 180,E1 7731.628,E2 7731.628} C_VEL
LIN {X 0,Y 364.715,Z 712.445,A -85,B 0,C 180,E1 7730.279,E2 7730.279} C_VEL
LIN {X 0,Y 349.764,Z 845.542,A -85,B 0,C 180,E1 7728.502,E2 7728.502} C_VEL
LIN {X 0,Y 345.219,Z 870.42,A -85,B 0,C 180,E1 7728.107,E2 7728.107} C_VEL
LIN {X 0,Y 339.659,Z 892.698,A -85,B 0,C 180,E1 7727.658,E2 7727.658} C_VEL
LIN {X 0,Y 332.421,Z 915.227,A -85,B 0,C 180,E1 7727.05,E2 7727.05} C_VEL
LIN {X 0,Y 324.795,Z 934.987,A -85,B 0,C 180,E1 7726.376,E2 7726.376} C_VEL
LIN {X 0,Y 314.604,Z 957.19,A -85,B 0,C 180,E1 7725.417,E2 7725.417} C_VEL
LIN {X 0,Y 304.365,Z 976.38,A -85,B 0,C 180,E1 7724.372,E2 7724.372} C_VEL
LIN {X 0,Y 291.763,Z 996.875,A -85,B 0,C 180,E1 7722.971,E2 7722.971} C_VEL
LIN {X 0,Y 279.488,Z 1014.495,A -85,B 0,C 180,E1 7721.453,E2 7721.453} C_VEL
LIN {X 0,Y 264.882,Z 1033.019,A -85,B 0,C 180,E1 7719.418,E2 7719.418} C_VEL
LIN {X 0,Y 251.474,Z 1048.271,A -85,B 0,C 180,E1 7717.289,E2 7717.289} C_VEL
LIN {X 0,Y 236.052,Z 1063.998,A -85,B 0,C 180,E1 7714.456,E2 7714.456} C_VEL
LIN {X 0,Y 222.048,Z 1076.99,A -85,B 0,C 180,E1 7711.414,E2 7711.414} C_VEL
LIN {X 0,Y 206.593,Z 1090.012,A -85,B 0,C 180,E1 7707.368,E2 7707.368} C_VEL
LIN {X 0,Y 192.94,Z 1100.641,A -85,B 0,C 180,E1 7702.949,E2 7702.949} C_VEL
LIN {X 0,Y 178.812,Z 1110.819,A -85,B 0,C 180,E1 7697.099,E2 7697.099} C_VEL
LIN {X 0,Y 167.202,Z 1118.852,A -85,B 0,C 180,E1 7690.68,E2 7690.68} C_VEL
LIN {X 0,Y 157.387,Z 1125.394,A -85,B 0,C 180,E1 7683.118,E2 7683.118} C_VEL
LIN {X 0,Y 150.293,Z 1130.396,A -85,B 0,C 180,E1 7674.78,E2 7674.78} C_VEL
LIN {X 0,Y 146.001,Z 1133.678,A -85,B 0,C 180,E1 7665.899,E2 7665.899} C_VEL
LIN {X 0,Y 144.417,Z 1135.301,A -85,B 0,C 180,E1 7658.36,E2 7658.36} C_VEL
LIN {X 0,Y 144.055,Z 1135.949,A -85,B 0,C 180,E1 7650.795,E2 7650.795} C_VEL
LIN {X 0,Y 144.257,Z 1135.594,A -85,B 0,C 180,E1 7643.233,E2 7643.233} C_VEL
LIN {X 0,Y 145.735,Z 1133.951,A -85,B 0,C 180,E1 7634.887,E2 7634.887} C_VEL
LIN {X 0,Y 149.502,Z 1130.994,A -85,B 0,C 180,E1 7626.388,E2 7626.388} C_VEL
LIN {X 0,Y 156.594,Z 1126.009,A -85,B 0,C 180,E1 7617.564,E2 7617.564} C_VEL
LIN {X 0,Y 165.694,Z 1119.95,A -85,B 0,C 180,E1 7610.233,E2 7610.233} C_VEL
LIN {X 0,Y 177.725,Z 1111.701,A -85,B 0,C 180,E1 7603.345,E2 7603.345} C_VEL
LIN {X 0,Y 190.892,Z 1102.35,A -85,B 0,C 180,E1 7597.726,E2 7597.726} C_VEL
LIN {X 0,Y 205.067,Z 1091.403,A -85,B 0,C 180,E1 7593.001,E2 7593.001} C_VEL
LIN {X 0,Y 220.426,Z 1078.69,A -85,B 0,C 180,E1 7588.897,E2 7588.897} C_VEL
LIN {X 0,Y 235.146,Z 1065.109,A -85,B 0,C 180,E1 7585.648,E2 7585.648} C_VEL
LIN {X 0,Y 249.717,Z 1050.509,A -85,B 0,C 180,E1 7582.935,E2 7582.935} C_VEL
LIN {X 0,Y 264.178,Z 1034.179,A -85,B 0,C 180,E1 7580.61,E2 7580.61} C_VEL
LIN {X 0,Y 277.984,Z 1016.985,A -85,B 0,C 180,E1 7578.671,E2 7578.671} C_VEL
LIN {X 0,Y 291.22,Z 998.135,A -85,B 0,C 180,E1 7577.016,E2 7577.016} C_VEL
LIN {X 0,Y 303.693,Z 978.135,A -85,B 0,C 180,E1 7575.625,E2 7575.625} C_VEL
LIN {X 0,Y 314.055,Z 958.867,A -85,B 0,C 180,E1 7574.561,E2 7574.561} C_VEL
LIN {X 0,Y 324.075,Z 937.511,A -85,B 0,C 180,E1 7573.616,E2 7573.616} C_VEL
LIN {X 0,Y 332.33,Z 916.339,A -85,B 0,C 180,E1 7572.882,E2 7572.882} C_VEL
LIN {X 0,Y 339.793,Z 893.366,A -85,B 0,C 180,E1 7572.256,E2 7572.256} C_VEL
LIN {X 0,Y 345.467,Z 870.717,A -85,B 0,C 180,E1 7571.799,E2 7571.799} C_VEL
LIN {X 0,Y 350.003,Z 846.143,A -85,B 0,C 180,E1 7571.407,E2 7571.407} C_VEL
LIN {X 0,Y 361.831,Z 741.46,A -85,B 0,C 180,E1 7570.004,E2 7570.004} C_VEL
LIN {X 0,Y 365.052,Z 712.443,A -85,B 0,C 180,E1 7569.618,E2 7569.618} C_VEL
LIN {X 0,Y 363.757,Z 707.842,A -85,B 0,C 180,E1 7567.105,E2 7567.105} C_VEL
LIN {X 0,Y 363.002,Z 705.008,A -85,B 0,C 180,E1 7564.74,E2 7564.74} C_VEL
LIN {X 0,Y 362.707,Z 703.181,A -85,B 0,C 180,E1 7560.79,E2 7560.79} C_VEL
LIN {X 0,Y 363.076,Z 704.018,A -85,B 0,C 180,E1 7558.567,E2 7558.567} C_VEL
LIN {X 0,Y 364.198,Z 706.482,A -85,B 0,C 180,E1 7555.749,E2 7555.749} C_VEL
LIN {X 0,Y 365.495,Z 709.782,A -85,B 0,C 180,E1 7553.582,E2 7553.582} C_VEL
LIN {X 0,Y 350.147,Z 844.802,A -85,B 0,C 180,E1 7551.736,E2 7551.736} C_VEL
LIN {X 0,Y 345.542,Z 869.927,A -85,B 0,C 180,E1 7551.325,E2 7551.325} C_VEL
LIN {X 0,Y 345.419,Z 870.476,A -85,B 0,C 180,E1 7551.315,E2 7551.315} C_VEL
LIN {X 0,Y 343.544,Z 877.999,A -85,B 0,C 180,E1 7551.367,E2 7551.367} C_VEL
LIN {X 0,Y 337.377,Z 896.834,A -85,B 0,C 180,E1 7551.962,E2 7551.962} C_VEL
LIN {X 0,Y 334.888,Z 904.19,A -85,B 0,C 180,E1 7551.911,E2 7551.911} C_VEL
LIN {X 0,Y 326.298,Z 927.979,A -85,B 0,C 180,E1 7551.21,E2 7551.21} C_VEL
LIN {X 0,Y 317.385,Z 948.453,A -85,B 0,C 180,E1 7550.43,E2 7550.43} C_VEL
LIN {X 0,Y 305.753,Z 971.23,A -85,B 0,C 180,E1 7549.332,E2 7549.332} C_VEL
LIN {X 0,Y 294.694,Z 989.93,A -85,B 0,C 180,E1 7548.204,E2 7548.204} C_VEL
LIN {X 0,Y 280.528,Z 1010.905,A -85,B 0,C 180,E1 7546.604,E2 7546.604} C_VEL
LIN {X 0,Y 267.602,Z 1027.843,A -85,B 0,C 180,E1 7544.963,E2 7544.963} C_VEL
LIN {X 0,Y 251.674,Z 1046.403,A -85,B 0,C 180,E1 7542.664,E2 7542.664} C_VEL
LIN {X 0,Y 237.756,Z 1060.999,A -85,B 0,C 180,E1 7540.34,E2 7540.34} C_VEL
LIN {X 0,Y 221.395,Z 1076.5,A -85,B 0,C 180,E1 7537.122,E2 7537.122} C_VEL
LIN {X 0,Y 207.289,Z 1088.694,A -85,B 0,C 180,E1 7533.793,E2 7533.793} C_VEL
LIN {X 0,Y 190.419,Z 1102.075,A -85,B 0,C 180,E1 7528.861,E2 7528.861} C_VEL
LIN {X 0,Y 177.041,Z 1111.958,A -85,B 0,C 180,E1 7523.866,E2 7523.866} C_VEL
LIN {X 0,Y 163.5,Z 1121.433,A -85,B 0,C 180,E1 7517.212,E2 7517.212} C_VEL
LIN {X 0,Y 153.111,Z 1128.568,A -85,B 0,C 180,E1 7510.175,E2 7510.175} C_VEL
LIN {X 0,Y 143.961,Z 1135.041,A -85,B 0,C 180,E1 7500.929,E2 7500.929} C_VEL
LIN {X 0,Y 138.975,Z 1139.043,A -85,B 0,C 180,E1 7492.416,E2 7492.416} C_VEL
LIN {X 0,Y 136.371,Z 1141.945,A -85,B 0,C 180,E1 7482.707,E2 7482.707} C_VEL
LIN {X 0,Y 135.988,Z 1143.083,A -85,B 0,C 180,E1 7474.639,E2 7474.639} C_VEL
LIN {X 0,Y 136.03,Z 1143.261,A -85,B 0,C 180,E1 7468.545,E2 7468.545} C_VEL
LIN {X 0,Y 136.025,Z 1142.653,A -85,B 0,C 180,E1 7461.546,E2 7461.546} C_VEL
LIN {X 0,Y 137.058,Z 1140.932,A -85,B 0,C 180,E1 7453.47,E2 7453.47} C_VEL
LIN {X 0,Y 140.349,Z 1137.831,A -85,B 0,C 180,E1 7444.693,E2 7444.693} C_VEL
LIN {X 0,Y 147.228,Z 1132.591,A -85,B 0,C 180,E1 7435.216,E2 7435.216} C_VEL
LIN {X 0,Y 155.914,Z 1126.544,A -85,B 0,C 180,E1 7427.672,E2 7427.672} C_VEL
LIN {X 0,Y 168.532,Z 1117.837,A -85,B 0,C 180,E1 7420.062,E2 7420.062} C_VEL
LIN {X 0,Y 180.902,Z 1109.016,A -85,B 0,C 180,E1 7414.557,E2 7414.557} C_VEL
LIN {X 0,Y 196.837,Z 1096.958,A -85,B 0,C 180,E1 7409.105,E2 7409.105} C_VEL
LIN {X 0,Y 211.119,Z 1085.28,A -85,B 0,C 180,E1 7405.229,E2 7405.229} C_VEL
LIN {X 0,Y 227.862,Z 1070.314,A -85,B 0,C 180,E1 7401.52,E2 7401.52} C_VEL
LIN {X 0,Y 242.022,Z 1056.39,A -85,B 0,C 180,E1 7398.898,E2 7398.898} C_VEL
LIN {X 0,Y 258.374,Z 1038.535,A -85,B 0,C 180,E1 7396.311,E2 7396.311} C_VEL
LIN {X 0,Y 272.061,Z 1021.846,A -85,B 0,C 180,E1 7394.435,E2 7394.435} C_VEL
LIN {X 0,Y 286.167,Z 1002.441,A -85,B 0,C 180,E1 7392.717,E2 7392.717} C_VEL
LIN {X 0,Y 297.893,Z 984.263,A -85,B 0,C 180,E1 7391.445,E2 7391.445} C_VEL
LIN {X 0,Y 309.914,Z 962.909,A -85,B 0,C 180,E1 7390.25,E2 7390.25} C_VEL
LIN {X 0,Y 319.247,Z 943.757,A -85,B 0,C 180,E1 7389.392,E2 7389.392} C_VEL
LIN {X 0,Y 329.118,Z 919.846,A -85,B 0,C 180,E1 7388.544,E2 7388.544} C_VEL
LIN {X 0,Y 336.211,Z 899.025,A -85,B 0,C 180,E1 7387.968,E2 7387.968} C_VEL
LIN {X 0,Y 343.008,Z 873.836,A -85,B 0,C 180,E1 7387.439,E2 7387.439} C_VEL
LIN {X 0,Y 347.546,Z 851.249,A -85,B 0,C 180,E1 7387.071,E2 7387.071} C_VEL
LIN {X 0,Y 351.802,Z 818.201,A -85,B 0,C 180,E1 7386.61,E2 7386.61} C_VEL
LIN {X 0,Y 363.445,Z 715.695,A -85,B 0,C 180,E1 7385.234,E2 7385.234} C_VEL
LIN {X 0,Y 362.49,Z 713.196,A -85,B 0,C 180,E1 7383.321,E2 7383.321} C_VEL
LIN {X 0,Y 361.542,Z 710.807,A -85,B 0,C 180,E1 7380,E2 7380} C_VEL
LIN {X 0,Y 361.341,Z 711.078,A -85,B 0,C 180,E1 7377.938,E2 7377.938} C_VEL
LIN {X 0,Y 361.788,Z 713.315,A -85,B 0,C 180,E1 7374.608,E2 7374.608} C_VEL
LIN {X 0,Y 362.818,Z 717.165,A -85,B 0,C 180,E1 7371.92,E2 7371.92} C_VEL
LIN {X 0,Y 363.023,Z 718.28,A -85,B 0,C 180,E1 7371.456,E2 7371.456} C_VEL
LIN {X 0,Y 348.471,Z 845.566,A -85,B 0,C 180,E1 7369.8,E2 7369.8} C_VEL
LIN {X 0,Y 343.89,Z 870.332,A -85,B 0,C 180,E1 7369.422,E2 7369.422} C_VEL
LIN {X 0,Y 338.333,Z 892.379,A -85,B 0,C 180,E1 7368.999,E2 7368.999} C_VEL
LIN {X 0,Y 331.189,Z 914.498,A -85,B 0,C 180,E1 7368.436,E2 7368.436} C_VEL
LIN {X 0,Y 323.293,Z 934.773,A -85,B 0,C 180,E1 7367.78,E2 7367.78} C_VEL
LIN {X 0,Y 312.683,Z 957.585,A -85,B 0,C 180,E1 7366.838,E2 7366.838} C_VEL
LIN {X 0,Y 302.171,Z 976.975,A -85,B 0,C 180,E1 7365.824,E2 7365.824} C_VEL
LIN {X 0,Y 289.509,Z 997.19,A -85,B 0,C 180,E1 7364.494,E2 7364.494} C_VEL
LIN {X 0,Y 277.029,Z 1014.793,A -85,B 0,C 180,E1 7363.034,E2 7363.034} C_VEL
LIN {X 0,Y 262.149,Z 1033.287,A -85,B 0,C 180,E1 7361.072,E2 7361.072} C_VEL
LIN {X 0,Y 248.454,Z 1048.537,A -85,B 0,C 180,E1 7359.012,E2 7359.012} C_VEL
LIN {X 0,Y 232.665,Z 1064.24,A -85,B 0,C 180,E1 7356.26,E2 7356.26} C_VEL
LIN {X 0,Y 218.271,Z 1077.228,A -85,B 0,C 180,E1 7353.29,E2 7353.29} C_VEL
LIN {X 0,Y 202.315,Z 1090.242,A -85,B 0,C 180,E1 7349.312,E2 7349.312} C_VEL
LIN {X 0,Y 188.136,Z 1100.867,A -85,B 0,C 180,E1 7344.932,E2 7344.932} C_VEL
LIN {X 0,Y 173.962,Z 1110.642,A -85,B 0,C 180,E1 7339.351,E2 7339.351} C_VEL
LIN {X 0,Y 161.608,Z 1118.726,A -85,B 0,C 180,E1 7332.89,E2 7332.89} C_VEL
LIN {X 0,Y 151.024,Z 1125.362,A -85,B 0,C 180,E1 7325.17,E2 7325.17} C_VEL
LIN {X 0,Y 143.424,Z 1130.264,A -85,B 0,C 180,E1 7316.828,E2 7316.828} C_VEL
LIN {X 0,Y 138.389,Z 1133.782,A -85,B 0,C 180,E1 7307.232,E2 7307.232} C_VEL
LIN {X 0,Y 136.522,Z 1135.447,A -85,B 0,C 180,E1 7299.272,E2 7299.272} C_VEL
LIN {X 0,Y 136.06,Z 1136.115,A -85,B 0,C 180,E1 7291.685,E2 7291.685} C_VEL
LIN {X 0,Y 136.169,Z 1135.935,A -85,B 0,C 180,E1 7284.522,E2 7284.522} C_VEL
LIN {X 0,Y 137.586,Z 1134.489,A -85,B 0,C 180,E1 7275.264,E2 7275.264} C_VEL
LIN {X 0,Y 141.157,Z 1131.804,A -85,B 0,C 180,E1 7266.629,E2 7266.629} C_VEL
LIN {X 0,Y 148.283,Z 1127.212,A -85,B 0,C 180,E1 7257.354,E2 7257.354} C_VEL
LIN {X 0,Y 157.771,Z 1121.214,A -85,B 0,C 180,E1 7249.51,E2 7249.51} C_VEL
LIN {X 0,Y 170.885,Z 1112.816,A -85,B 0,C 180,E1 7242.003,E2 7242.003} C_VEL
LIN {X 0,Y 184.007,Z 1103.92,A -85,B 0,C 180,E1 7236.464,E2 7236.464} C_VEL
LIN {X 0,Y 200.014,Z 1092.191,A -85,B 0,C 180,E1 7231.257,E2 7231.257} C_VEL
LIN {X 0,Y 215.054,Z 1080.193,A -85,B 0,C 180,E1 7227.37,E2 7227.37} C_VEL
LIN {X 0,Y 230.932,Z 1066.109,A -85,B 0,C 180,E1 7223.993,E2 7223.993} C_VEL
LIN {X 0,Y 245.828,Z 1051.596,A -85,B 0,C 180,E1 7221.338,E2 7221.338} C_VEL
LIN {X 0,Y 261.184,Z 1034.74,A -85,B 0,C 180,E1 7218.987,E2 7218.987} C_VEL
LIN {X 0,Y 275.262,Z 1017.583,A -85,B 0,C 180,E1 7217.112,E2 7217.112} C_VEL
LIN {X 0,Y 288.518,Z 999.103,A -85,B 0,C 180,E1 7215.54,E2 7215.54} C_VEL
LIN {X 0,Y 301.176,Z 979.294,A -85,B 0,C 180,E1 7214.203,E2 7214.203} C_VEL
LIN {X 0,Y 312.137,Z 959.252,A -85,B 0,C 180,E1 7213.137,E2 7213.137} C_VEL
LIN {X 0,Y 322.286,Z 937.982,A -85,B 0,C 180,E1 7212.234,E2 7212.234} C_VEL
LIN {X 0,Y 330.642,Z 916.872,A -85,B 0,C 180,E1 7211.533,E2 7211.533} C_VEL
LIN {X 0,Y 338.178,Z 894.137,A -85,B 0,C 180,E1 7210.938,E2 7210.938} C_VEL
LIN {X 0,Y 344.035,Z 871.12,A -85,B 0,C 180,E1 7210.492,E2 7210.492} C_VEL
LIN {X 0,Y 348.636,Z 846.769,A -85,B 0,C 180,E1 7210.118,E2 7210.118} C_VEL
LIN {X 0,Y 358.594,Z 760.721,A -85,B 0,C 180,E1 7208.99,E2 7208.99} C_VEL
LIN {X 0,Y 363.36,Z 718.383,A -85,B 0,C 180,E1 7208.437,E2 7208.437} C_VEL
LIN {X 0,Y 362.459,Z 714.97,A -85,B 0,C 180,E1 7206.335,E2 7206.335} C_VEL
LIN {X 0,Y 361.948,Z 712.804,A -85,B 0,C 180,E1 7204.436,E2 7204.436} C_VEL
LIN {X 0,Y 361.733,Z 711.122,A -85,B 0,C 180,E1 7200.792,E2 7200.792} C_VEL
LIN {X 0,Y 362.055,Z 711.908,A -85,B 0,C 180,E1 7198.7,E2 7198.7} C_VEL
LIN {X 0,Y 363.083,Z 714.279,A -85,B 0,C 180,E1 7195.973,E2 7195.973} C_VEL
LIN {X 0,Y 363.709,Z 716.217,A -85,B 0,C 180,E1 7194.747,E2 7194.747} C_VEL
LIN {X 0,Y 348.868,Z 844.821,A -85,B 0,C 180,E1 7193.033,E2 7193.033} C_VEL
LIN {X 0,Y 344.209,Z 869.96,A -85,B 0,C 180,E1 7192.638,E2 7192.638} C_VEL
LIN {X 0,Y 338.551,Z 892.348,A -85,B 0,C 180,E1 7192.196,E2 7192.196} C_VEL
LIN {X 0,Y 334.888,Z 904.19,A -85,B 0,C 180,E1 7191.911,E2 7191.911} C_VEL
LIN {X 0,Y 332.288,Z 911.578,A -85,B 0,C 180,E1 7191.883,E2 7191.883} C_VEL
LIN {X 0,Y 324.331,Z 929.877,A -85,B 0,C 180,E1 7192.368,E2 7192.368} C_VEL
LIN {X 0,Y 321.248,Z 936.872,A -85,B 0,C 180,E1 7192.302,E2 7192.302} C_VEL
LIN {X 0,Y 310.935,Z 958.558,A -85,B 0,C 180,E1 7191.436,E2 7191.436} C_VEL
LIN {X 0,Y 300.132,Z 978.237,A -85,B 0,C 180,E1 7190.446,E2 7190.446} C_VEL
LIN {X 0,Y 287.101,Z 998.753,A -85,B 0,C 180,E1 7189.152,E2 7189.152} C_VEL
LIN {X 0,Y 274.701,Z 1016.046,A -85,B 0,C 180,E1 7187.776,E2 7187.776} C_VEL
LIN {X 0,Y 259.172,Z 1035.172,A -85,B 0,C 180,E1 7185.842,E2 7185.842} C_VEL
LIN {X 0,Y 244.721,Z 1051.081,A -85,B 0,C 180,E1 7183.776,E2 7183.776} C_VEL
LIN {X 0,Y 228.352,Z 1067.179,A -85,B 0,C 180,E1 7181.051,E2 7181.051} C_VEL
LIN {X 0,Y 213.392,Z 1080.529,A -85,B 0,C 180,E1 7178.09,E2 7178.09} C_VEL
LIN {X 0,Y 196.68,Z 1094.03,A -85,B 0,C 180,E1 7174.074,E2 7174.074} C_VEL
LIN {X 0,Y 181.849,Z 1105.059,A -85,B 0,C 180,E1 7169.611,E2 7169.611} C_VEL
LIN {X 0,Y 166.433,Z 1115.657,A -85,B 0,C 180,E1 7163.614,E2 7163.614} C_VEL
LIN {X 0,Y 154.072,Z 1123.752,A -85,B 0,C 180,E1 7157.168,E2 7157.168} C_VEL
LIN {X 0,Y 142.532,Z 1131.13,A -85,B 0,C 180,E1 7148.635,E2 7148.635} C_VEL
LIN {X 0,Y 135.095,Z 1136.111,A -85,B 0,C 180,E1 7140.218,E2 7140.218} C_VEL
LIN {X 0,Y 129.767,Z 1140.27,A -85,B 0,C 180,E1 7129.349,E2 7129.349} C_VEL
LIN {X 0,Y 128.148,Z 1142.212,A -85,B 0,C 180,E1 7120.538,E2 7120.538} C_VEL
LIN {X 0,Y 128.001,Z 1142.948,A -85,B 0,C 180,E1 7113.583,E2 7113.583} C_VEL
LIN {X 0,Y 128.016,Z 1143.014,A -85,B 0,C 180,E1 7107.762,E2 7107.762} C_VEL
LIN {X 0,Y 128.078,Z 1142.369,A -85,B 0,C 180,E1 7100.564,E2 7100.564} C_VEL
LIN {X 0,Y 129.42,Z 1140.562,A -85,B 0,C 180,E1 7091.859,E2 7091.859} C_VEL
LIN {X 0,Y 133.716,Z 1137.112,A -85,B 0,C 180,E1 7081.894,E2 7081.894} C_VEL
LIN {X 0,Y 141.529,Z 1131.703,A -85,B 0,C 180,E1 7072.305,E2 7072.305} C_VEL
LIN {X 0,Y 152.468,Z 1124.737,A -85,B 0,C 180,E1 7063.831,E2 7063.831} C_VEL
LIN {X 0,Y 165.168,Z 1116.367,A -85,B 0,C 180,E1 7056.955,E2 7056.955} C_VEL
LIN {X 0,Y 179.806,Z 1106.426,A -85,B 0,C 180,E1 7051.086,E2 7051.086} C_VEL
LIN {X 0,Y 195.21,Z 1094.974,A -85,B 0,C 180,E1 7046.314,E2 7046.314} C_VEL
LIN {X 0,Y 211.756,Z 1081.741,A -85,B 0,C 180,E1 7042.256,E2 7042.256} C_VEL
LIN {X 0,Y 227.493,Z 1067.722,A -85,B 0,C 180,E1 7039.093,E2 7039.093} C_VEL
LIN {X 0,Y 243.835,Z 1051.729,A -85,B 0,C 180,E1 7036.349,E2 7036.349} C_VEL
LIN {X 0,Y 258.421,Z 1035.697,A -85,B 0,C 180,E1 7034.246,E2 7034.246} C_VEL
LIN {X 0,Y 273.322,Z 1017.498,A -85,B 0,C 180,E1 7032.374,E2 7032.374} C_VEL
LIN {X 0,Y 286.163,Z 999.663,A -85,B 0,C 180,E1 7030.931,E2 7030.931} C_VEL
LIN {X 0,Y 299.186,Z 979.337,A -85,B 0,C 180,E1 7029.631,E2 7029.631} C_VEL
LIN {X 0,Y 310.156,Z 959.449,A -85,B 0,C 180,E1 7028.619,E2 7028.619} C_VEL
LIN {X 0,Y 320.397,Z 938.147,A -85,B 0,C 180,E1 7027.755,E2 7027.755} C_VEL
LIN {X 0,Y 329.007,Z 916.6,A -85,B 0,C 180,E1 7027.07,E2 7027.07} C_VEL
LIN {X 0,Y 336.737,Z 893.38,A -85,B 0,C 180,E1 7026.489,E2 7026.489} C_VEL
LIN {X 0,Y 342.596,Z 870.569,A -85,B 0,C 180,E1 7026.057,E2 7026.057} C_VEL
LIN {X 0,Y 347.296,Z 845.876,A -85,B 0,C 180,E1 7025.683,E2 7025.683} C_VEL
LIN {X 0,Y 357.35,Z 760.775,A -85,B 0,C 180,E1 7024.568,E2 7024.568} C_VEL
LIN {X 0,Y 361.809,Z 722.117,A -85,B 0,C 180,E1 7024.041,E2 7024.041} C_VEL
LIN {X 0,Y 361.119,Z 720.445,A -85,B 0,C 180,E1 7022.38,E2 7022.38} C_VEL
LIN {X 0,Y 360.521,Z 718.668,A -85,B 0,C 180,E1 7019.682,E2 7019.682} C_VEL
LIN {X 0,Y 360.361,Z 719.307,A -85,B 0,C 180,E1 7017.434,E2 7017.434} C_VEL
LIN {X 0,Y 360.764,Z 721.232,A -85,B 0,C 180,E1 7014.752,E2 7014.752} C_VEL
LIN {X 0,Y 361.479,Z 724.154,A -85,B 0,C 180,E1 7012.644,E2 7012.644} C_VEL
LIN {X 0,Y 347.358,Z 845.59,A -85,B 0,C 180,E1 7011.107,E2 7011.107} C_VEL
LIN {X 0,Y 342.702,Z 870.427,A -85,B 0,C 180,E1 7010.744,E2 7010.744} C_VEL
LIN {X 0,Y 337.078,Z 892.485,A -85,B 0,C 180,E1 7010.342,E2 7010.342} C_VEL
LIN {X 0,Y 329.682,Z 915.046,A -85,B 0,C 180,E1 7009.795,E2 7009.795} C_VEL
LIN {X 0,Y 321.695,Z 935.257,A -85,B 0,C 180,E1 7009.171,E2 7009.171} C_VEL
LIN {X 0,Y 311.421,Z 957.086,A -85,B 0,C 180,E1 7008.316,E2 7008.316} C_VEL
LIN {X 0,Y 300.766,Z 976.533,A -85,B 0,C 180,E1 7007.353,E2 7007.353} C_VEL
LIN {X 0,Y 287.463,Z 997.506,A -85,B 0,C 180,E1 7006.039,E2 7006.039} C_VEL
LIN {X 0,Y 274.784,Z 1015.091,A -85,B 0,C 180,E1 7004.643,E2 7004.643} C_VEL
LIN {X 0,Y 259.64,Z 1033.557,A -85,B 0,C 180,E1 7002.76,E2 7002.76} C_VEL
LIN {X 0,Y 244.813,Z 1049.707,A -85,B 0,C 180,E1 7000.644,E2 7000.644} C_VEL
LIN {X 0,Y 229.516,Z 1064.482,A -85,B 0,C 180,E1 6998.116,E2 6998.116} C_VEL
LIN {X 0,Y 214.674,Z 1077.52,A -85,B 0,C 180,E1 6995.216,E2 6995.216} C_VEL
LIN {X 0,Y 198.279,Z 1090.469,A -85,B 0,C 180,E1 6991.338,E2 6991.338} C_VEL
LIN {X 0,Y 183.41,Z 1101.207,A -85,B 0,C 180,E1 6986.964,E2 6986.964} C_VEL
LIN {X 0,Y 168.121,Z 1111.26,A -85,B 0,C 180,E1 6981.18,E2 6981.18} C_VEL
LIN {X 0,Y 154.644,Z 1119.634,A -85,B 0,C 180,E1 6974.291,E2 6974.291} C_VEL
LIN {X 0,Y 143.58,Z 1126.071,A -85,B 0,C 180,E1 6966.295,E2 6966.295} C_VEL
LIN {X 0,Y 135.409,Z 1131.016,A -85,B 0,C 180,E1 6957.247,E2 6957.247} C_VEL
LIN {X 0,Y 130.367,Z 1134.211,A -85,B 0,C 180,E1 6947.405,E2 6947.405} C_VEL
LIN {X 0,Y 128.424,Z 1135.853,A -85,B 0,C 180,E1 6938.507,E2 6938.507} C_VEL
LIN {X 0,Y 128.065,Z 1136.411,A -85,B 0,C 180,E1 6930,E2 6930} C_VEL
LIN {X 0,Y 128.425,Z 1135.874,A -85,B 0,C 180,E1 6921.417,E2 6921.417} C_VEL
LIN {X 0,Y 130.338,Z 1134.266,A -85,B 0,C 180,E1 6912.591,E2 6912.591} C_VEL
LIN {X 0,Y 135.358,Z 1131.094,A -85,B 0,C 180,E1 6902.742,E2 6902.742} C_VEL
LIN {X 0,Y 143.512,Z 1126.191,A -85,B 0,C 180,E1 6893.685,E2 6893.685} C_VEL
LIN {X 0,Y 154.558,Z 1119.786,A -85,B 0,C 180,E1 6885.678,E2 6885.678} C_VEL
LIN {X 0,Y 167.396,Z 1111.843,A -85,B 0,C 180,E1 6879.057,E2 6879.057} C_VEL
LIN {X 0,Y 182.063,Z 1102.327,A -85,B 0,C 180,E1 6873.406,E2 6873.406} C_VEL
LIN {X 0,Y 197.878,Z 1090.945,A -85,B 0,C 180,E1 6868.688,E2 6868.688} C_VEL
LIN {X 0,Y 213.835,Z 1078.467,A -85,B 0,C 180,E1 6864.886,E2 6864.886} C_VEL
LIN {X 0,Y 229.419,Z 1064.825,A -85,B 0,C 180,E1 6861.823,E2 6861.823} C_VEL
LIN {X 0,Y 245.58,Z 1049.196,A -85,B 0,C 180,E1 6859.16,E2 6859.16} C_VEL
LIN {X 0,Y 259.99,Z 1033.495,A -85,B 0,C 180,E1 6857.117,E2 6857.117} C_VEL
LIN {X 0,Y 275.147,Z 1015.014,A -85,B 0,C 180,E1 6855.239,E2 6855.239} C_VEL
LIN {X 0,Y 287.834,Z 997.422,A -85,B 0,C 180,E1 6853.846,E2 6853.846} C_VEL
LIN {X 0,Y 301.148,Z 976.424,A -85,B 0,C 180,E1 6852.535,E2 6852.535} C_VEL
LIN {X 0,Y 311.808,Z 956.952,A -85,B 0,C 180,E1 6851.574,E2 6851.574} C_VEL
LIN {X 0,Y 322.557,Z 933.961,A -85,B 0,C 180,E1 6850.682,E2 6850.682} C_VEL
LIN {X 0,Y 330.553,Z 913.573,A -85,B 0,C 180,E1 6850.064,E2 6850.064} C_VEL
LIN {X 0,Y 338.288,Z 889.271,A -85,B 0,C 180,E1 6849.496,E2 6849.496} C_VEL
LIN {X 0,Y 343.737,Z 867.348,A -85,B 0,C 180,E1 6849.109,E2 6849.109} C_VEL
LIN {X 0,Y 348.121,Z 842.454,A -85,B 0,C 180,E1 6848.754,E2 6848.754} C_VEL
LIN {X 0,Y 361.824,Z 724.425,A -85,B 0,C 180,E1 6847.263,E2 6847.263} C_VEL
LIN {X 0,Y 360.972,Z 720.78,A -85,B 0,C 180,E1 6844.448,E2 6844.448} C_VEL
LIN {X 0,Y 360.774,Z 719.054,A -85,B 0,C 180,E1 6840.635,E2 6840.635} C_VEL
LIN {X 0,Y 361.145,Z 720.093,A -85,B 0,C 180,E1 6838.413,E2 6838.413} C_VEL
LIN {X 0,Y 362.043,Z 722.298,A -85,B 0,C 180,E1 6836.041,E2 6836.041} C_VEL
LIN {X 0,Y 362.066,Z 722.721,A -85,B 0,C 180,E1 6835.922,E2 6835.922} C_VEL
LIN {X 0,Y 347.754,Z 844.948,A -85,B 0,C 180,E1 6834.338,E2 6834.338} C_VEL
LIN {X 0,Y 343.03,Z 870.113,A -85,B 0,C 180,E1 6833.958,E2 6833.958} C_VEL
LIN {X 0,Y 337.267,Z 892.642,A -85,B 0,C 180,E1 6833.535,E2 6833.535} C_VEL
LIN {X 0,Y 329.935,Z 914.971,A -85,B 0,C 180,E1 6832.986,E2 6832.986} C_VEL
LIN {X 0,Y 322.305,Z 934.334,A -85,B 0,C 180,E1 6832.391,E2 6832.391} C_VEL
LIN {X 0,Y 321.248,Z 936.872,A -85,B 0,C 180,E1 6832.302,E2 6832.302} C_VEL
LIN {X 0,Y 318.036,Z 943.934,A -85,B 0,C 180,E1 6832.222,E2 6832.222} C_VEL
LIN {X 0,Y 308.424,Z 961.496,A -85,B 0,C 180,E1 6832.599,E2 6832.599} C_VEL
LIN {X 0,Y 304.529,Z 968.164,A -85,B 0,C 180,E1 6832.473,E2 6832.473} C_VEL
LIN {X 0,Y 292.738,Z 987.782,A -85,B 0,C 180,E1 6831.431,E2 6831.431} C_VEL
LIN {X 0,Y 279.084,Z 1007.82,A -85,B 0,C 180,E1 6830.097,E2 6830.097} C_VEL
LIN {X 0,Y 265.227,Z 1025.561,A -85,B 0,C 180,E1 6828.576,E2 6828.576} C_VEL
LIN {X 0,Y 249.731,Z 1043.327,A -85,B 0,C 180,E1 6826.642,E2 6826.642} C_VEL
LIN {X 0,Y 234.14,Z 1059.12,A -85,B 0,C 180,E1 6824.393,E2 6824.393} C_VEL
LIN {X 0,Y 217.002,Z 1074.773,A -85,B 0,C 180,E1 6821.462,E2 6821.462} C_VEL
LIN {X 0,Y 201.335,Z 1087.583,A -85,B 0,C 180,E1 6818.234,E2 6818.234} C_VEL
LIN {X 0,Y 183.919,Z 1100.573,A -85,B 0,C 180,E1 6813.771,E2 6813.771} C_VEL
LIN {X 0,Y 169.189,Z 1110.572,A -85,B 0,C 180,E1 6808.975,E2 6808.975} C_VEL
LIN {X 0,Y 153.745,Z 1120.385,A -85,B 0,C 180,E1 6802.314,E2 6802.314} C_VEL
LIN {X 0,Y 141.47,Z 1127.753,A -85,B 0,C 180,E1 6794.974,E2 6794.974} C_VEL
LIN {X 0,Y 130.446,Z 1134.394,A -85,B 0,C 180,E1 6785.092,E2 6785.092} C_VEL
LIN {X 0,Y 124.068,Z 1138.545,A -85,B 0,C 180,E1 6775.493,E2 6775.493} C_VEL
LIN {X 0,Y 120.58,Z 1141.521,A -85,B 0,C 180,E1 6764.405,E2 6764.405} C_VEL
LIN {X 0,Y 119.987,Z 1142.662,A -85,B 0,C 180,E1 6755.26,E2 6755.26} C_VEL
LIN {X 0,Y 120.032,Z 1142.846,A -85,B 0,C 180,E1 6748.445,E2 6748.445} C_VEL
LIN {X 0,Y 120.058,Z 1142.302,A -85,B 0,C 180,E1 6740.895,E2 6740.895} C_VEL
LIN {X 0,Y 121.515,Z 1140.503,A -85,B 0,C 180,E1 6731.282,E2 6731.282} C_VEL
LIN {X 0,Y 125.955,Z 1137.232,A -85,B 0,C 180,E1 6721.037,E2 6721.037} C_VEL
LIN {X 0,Y 134.409,Z 1131.891,A -85,B 0,C 180,E1 6710.778,E2 6710.778} C_VEL
LIN {X 0,Y 145.18,Z 1125.479,A -85,B 0,C 180,E1 6702.529,E2 6702.529} C_VEL
LIN {X 0,Y 159.005,Z 1116.972,A -85,B 0,C 180,E1 6695.165,E2 6695.165} C_VEL
LIN {X 0,Y 173.474,Z 1107.628,A -85,B 0,C 180,E1 6689.5,E2 6689.5} C_VEL
LIN {X 0,Y 190.103,Z 1095.909,A -85,B 0,C 180,E1 6684.503,E2 6684.503} C_VEL
LIN {X 0,Y 206.265,Z 1083.517,A -85,B 0,C 180,E1 6680.676,E2 6680.676} C_VEL
LIN {X 0,Y 223.196,Z 1069.036,A -85,B 0,C 180,E1 6677.404,E2 6677.404} C_VEL
LIN {X 0,Y 238.974,Z 1054.17,A -85,B 0,C 180,E1 6674.865,E2 6674.865} C_VEL
LIN {X 0,Y 254.667,Z 1037.514,A -85,B 0,C 180,E1 6672.702,E2 6672.702} C_VEL
LIN {X 0,Y 268.907,Z 1020.714,A -85,B 0,C 180,E1 6670.993,E2 6670.993} C_VEL
LIN {X 0,Y 283.321,Z 1001.366,A -85,B 0,C 180,E1 6669.456,E2 6669.456} C_VEL
LIN {X 0,Y 296.037,Z 982.098,A -85,B 0,C 180,E1 6668.255,E2 6668.255} C_VEL
LIN {X 0,Y 307.911,Z 961.199,A -85,B 0,C 180,E1 6667.222,E2 6667.222} C_VEL
LIN {X 0,Y 317.963,Z 940.85,A -85,B 0,C 180,E1 6666.423,E2 6666.423} C_VEL
LIN {X 0,Y 327.105,Z 918.735,A -85,B 0,C 180,E1 6665.737,E2 6665.737} C_VEL
LIN {X 0,Y 334.596,Z 897.002,A -85,B 0,C 180,E1 6665.206,E2 6665.206} C_VEL
LIN {X 0,Y 341.079,Z 872.938,A -85,B 0,C 180,E1 6664.761,E2 6664.761} C_VEL
LIN {X 0,Y 345.864,Z 849.274,A -85,B 0,C 180,E1 6664.413,E2 6664.413} C_VEL
LIN {X 0,Y 351.036,Z 808.137,A -85,B 0,C 180,E1 6663.885,E2 6663.885} C_VEL
LIN {X 0,Y 360.309,Z 728.82,A -85,B 0,C 180,E1 6662.863,E2 6662.863} C_VEL
LIN {X 0,Y 359.545,Z 726.614,A -85,B 0,C 180,E1 6659.681,E2 6659.681} C_VEL
LIN {X 0,Y 359.383,Z 727.276,A -85,B 0,C 180,E1 6657.434,E2 6657.434} C_VEL
LIN {X 0,Y 359.726,Z 729.041,A -85,B 0,C 180,E1 6654.977,E2 6654.977} C_VEL
LIN {X 0,Y 360.011,Z 730.738,A -85,B 0,C 180,E1 6653.83,E2 6653.83} C_VEL
LIN {X 0,Y 346.427,Z 845.615,A -85,B 0,C 180,E1 6652.422,E2 6652.422} C_VEL
LIN {X 0,Y 341.728,Z 870.391,A -85,B 0,C 180,E1 6652.077,E2 6652.077} C_VEL
LIN {X 0,Y 336.072,Z 892.364,A -85,B 0,C 180,E1 6651.698,E2 6651.698} C_VEL
LIN {X 0,Y 328.486,Z 915.259,A -85,B 0,C 180,E1 6651.175,E2 6651.175} C_VEL
LIN {X 0,Y 320.29,Z 935.742,A -85,B 0,C 180,E1 6650.576,E2 6650.576} C_VEL
LIN {X 0,Y 309.898,Z 957.481,A -85,B 0,C 180,E1 6649.767,E2 6649.767} C_VEL
LIN {X 0,Y 299.112,Z 976.896,A -85,B 0,C 180,E1 6648.853,E2 6648.853} C_VEL
LIN {X 0,Y 286.091,Z 997.158,A -85,B 0,C 180,E1 6647.65,E2 6647.65} C_VEL
LIN {X 0,Y 273.217,Z 1014.785,A -85,B 0,C 180,E1 6646.326,E2 6646.326} C_VEL
LIN {X 0,Y 257.81,Z 1033.325,A -85,B 0,C 180,E1 6644.534,E2 6644.534} C_VEL
LIN {X 0,Y 242.42,Z 1049.79,A -85,B 0,C 180,E1 6642.476,E2 6642.476} C_VEL
LIN {X 0,Y 226.616,Z 1064.725,A -85,B 0,C 180,E1 6640.021,E2 6640.021} C_VEL
LIN {X 0,Y 210.632,Z 1078.396,A -85,B 0,C 180,E1 6637.064,E2 6637.064} C_VEL
LIN {X 0,Y 193.716,Z 1091.261,A -85,B 0,C 180,E1 6633.248,E2 6633.248} C_VEL
LIN {X 0,Y 177.795,Z 1102.331,A -85,B 0,C 180,E1 6628.741,E2 6628.741} C_VEL
LIN {X 0,Y 162.465,Z 1111.877,A -85,B 0,C 180,E1 6623.139,E2 6623.139} C_VEL
LIN {X 0,Y 148.341,Z 1120.158,A -85,B 0,C 180,E1 6616.157,E2 6616.157} C_VEL
LIN {X 0,Y 136.643,Z 1126.535,A -85,B 0,C 180,E1 6607.929,E2 6607.929} C_VEL
LIN {X 0,Y 127.616,Z 1131.539,A -85,B 0,C 180,E1 6598.042,E2 6598.042} C_VEL
LIN {X 0,Y 122.506,Z 1134.532,A -85,B 0,C 180,E1 6588.069,E2 6588.069} C_VEL
LIN {X 0,Y 120.376,Z 1136.194,A -85,B 0,C 180,E1 6578.118,E2 6578.118} C_VEL
LIN {X 0,Y 120.061,Z 1136.612,A -85,B 0,C 180,E1 6569.523,E2 6569.523} C_VEL
LIN {X 0,Y 120.53,Z 1136.031,A -85,B 0,C 180,E1 6560.45,E2 6560.45} C_VEL
LIN {X 0,Y 122.814,Z 1134.369,A -85,B 0,C 180,E1 6550.994,E2 6550.994} C_VEL
LIN {X 0,Y 128.514,Z 1131.126,A -85,B 0,C 180,E1 6540.623,E2 6540.623} C_VEL
LIN {X 0,Y 137.48,Z 1126.157,A -85,B 0,C 180,E1 6531.283,E2 6531.283} C_VEL
LIN {X 0,Y 149.396,Z 1119.672,A -85,B 0,C 180,E1 6523.153,E2 6523.153} C_VEL
LIN {X 0,Y 163.261,Z 1111.527,A -85,B 0,C 180,E1 6516.447,E2 6516.447} C_VEL
LIN {X 0,Y 179.165,Z 1101.542,A -85,B 0,C 180,E1 6510.745,E2 6510.745} C_VEL
LIN {X 0,Y 194.405,Z 1090.948,A -85,B 0,C 180,E1 6506.498,E2 6506.498} C_VEL
LIN {X 0,Y 211.365,Z 1078.01,A -85,B 0,C 180,E1 6502.709,E2 6502.709} C_VEL
LIN {X 0,Y 227.132,Z 1064.524,A -85,B 0,C 180,E1 6499.814,E2 6499.814} C_VEL
LIN {X 0,Y 243.923,Z 1048.533,A -85,B 0,C 180,E1 6497.231,E2 6497.231} C_VEL
LIN {X 0,Y 258.177,Z 1033.255,A -85,B 0,C 180,E1 6495.344,E2 6495.344} C_VEL
LIN {X 0,Y 273.596,Z 1014.699,A -85,B 0,C 180,E1 6493.558,E2 6493.558} C_VEL
LIN {X 0,Y 286.479,Z 997.064,A -85,B 0,C 180,E1 6492.236,E2 6492.236} C_VEL
LIN {X 0,Y 299.975,Z 975.97,A -85,B 0,C 180,E1 6490.995,E2 6490.995} C_VEL
LIN {X 0,Y 310.3,Z 957.335,A -85,B 0,C 180,E1 6490.124,E2 6490.124} C_VEL
LIN {X 0,Y 321.171,Z 934.431,A -85,B 0,C 180,E1 6489.28,E2 6489.28} C_VEL
LIN {X 0,Y 329.251,Z 914.106,A -85,B 0,C 180,E1 6488.696,E2 6488.696} C_VEL
LIN {X 0,Y 337.167,Z 889.626,A -85,B 0,C 180,E1 6488.153,E2 6488.153} C_VEL
LIN {X 0,Y 342.657,Z 867.837,A -85,B 0,C 180,E1 6487.788,E2 6487.788} C_VEL
LIN {X 0,Y 347.167,Z 842.742,A -85,B 0,C 180,E1 6487.446,E2 6487.446} C_VEL
LIN {X 0,Y 360.388,Z 730.778,A -85,B 0,C 180,E1 6486.052,E2 6486.052} C_VEL
LIN {X 0,Y 359.922,Z 728.574,A -85,B 0,C 180,E1 6484.142,E2 6484.142} C_VEL
LIN {X 0,Y 359.799,Z 726.995,A -85,B 0,C 180,E1 6480.637,E2 6480.637} C_VEL
LIN {X 0,Y 360.163,Z 728.094,A -85,B 0,C 180,E1 6478.409,E2 6478.409} C_VEL
LIN {X 0,Y 360.562,Z 729.353,A -85,B 0,C 180,E1 6477.106,E2 6477.106} C_VEL
LIN {X 0,Y 346.838,Z 844.967,A -85,B 0,C 180,E1 6475.651,E2 6475.651} C_VEL
LIN {X 0,Y 342.057,Z 870.165,A -85,B 0,C 180,E1 6475.289,E2 6475.289} C_VEL
LIN {X 0,Y 336.246,Z 892.659,A -85,B 0,C 180,E1 6474.889,E2 6474.889} C_VEL
LIN {X 0,Y 328.562,Z 915.726,A -85,B 0,C 180,E1 6474.351,E2 6474.351} C_VEL
LIN {X 0,Y 320.37,Z 936.136,A -85,B 0,C 180,E1 6473.75,E2 6473.75} C_VEL
LIN {X 0,Y 309.829,Z 958.169,A -85,B 0,C 180,E1 6472.923,E2 6472.923} C_VEL
LIN {X 0,Y 304.529,Z 968.164,A -85,B 0,C 180,E1 6472.473,E2 6472.473} C_VEL
LIN {X 0,Y 300.503,Z 974.822,A -85,B 0,C 180,E1 6472.331,E2 6472.331} C_VEL
LIN {X 0,Y 289.243,Z 991.441,A -85,B 0,C 180,E1 6472.594,E2 6472.594} C_VEL
LIN {X 0,Y 284.803,Z 997.676,A -85,B 0,C 180,E1 6472.412,E2 6472.412} C_VEL
LIN {X 0,Y 272.174,Z 1014.844,A -85,B 0,C 180,E1 6471.203,E2 6471.203} C_VEL
LIN {X 0,Y 256.278,Z 1033.946,A -85,B 0,C 180,E1 6469.484,E2 6469.484} C_VEL
LIN {X 0,Y 242.462,Z 1048.69,A -85,B 0,C 180,E1 6467.788,E2 6467.788} C_VEL
LIN {X 0,Y 225.317,Z 1065.133,A -85,B 0,C 180,E1 6465.336,E2 6465.336} C_VEL
LIN {X 0,Y 209.509,Z 1078.634,A -85,B 0,C 180,E1 6462.652,E2 6462.652} C_VEL
LIN {X 0,Y 191.197,Z 1092.74,A -85,B 0,C 180,E1 6458.848,E2 6458.848} C_VEL
LIN {X 0,Y 175.687,Z 1103.496,A -85,B 0,C 180,E1 6454.813,E2 6454.813} C_VEL
LIN {X 0,Y 158.559,Z 1114.385,A -85,B 0,C 180,E1 6449.052,E2 6449.052} C_VEL
LIN {X 0,Y 144.552,Z 1122.587,A -85,B 0,C 180,E1 6442.701,E2 6442.701} C_VEL
LIN {X 0,Y 130.512,Z 1130.433,A -85,B 0,C 180,E1 6433.592,E2 6433.592} C_VEL
LIN {X 0,Y 121.499,Z 1135.465,A -85,B 0,C 180,E1 6424.6,E2 6424.6} C_VEL
LIN {X 0,Y 114.647,Z 1139.722,A -85,B 0,C 180,E1 6412.566,E2 6412.566} C_VEL
LIN {X 0,Y 112.296,Z 1141.746,A -85,B 0,C 180,E1 6402.339,E2 6402.339} C_VEL
LIN {X 0,Y 111.998,Z 1142.527,A -85,B 0,C 180,E1 6394.096,E2 6394.096} C_VEL
LIN {X 0,Y 112.022,Z 1142.619,A -85,B 0,C 180,E1 6387.954,E2 6387.954} C_VEL
LIN {X 0,Y 112.123,Z 1142.017,A -85,B 0,C 180,E1 6379.726,E2 6379.726} C_VEL
LIN {X 0,Y 113.966,Z 1140.169,A -85,B 0,C 180,E1 6369.455,E2 6369.455} C_VEL
LIN {X 0,Y 119.451,Z 1136.679,A -85,B 0,C 180,E1 6358.173,E2 6358.173} C_VEL
LIN {X 0,Y 128.573,Z 1131.408,A -85,B 0,C 180,E1 6348.025,E2 6348.025} C_VEL
LIN {X 0,Y 140.886,Z 1124.635,A -85,B 0,C 180,E1 6339.322,E2 6339.322} C_VEL
LIN {X 0,Y 155.75,Z 1115.92,A -85,B 0,C 180,E1 6332.067,E2 6332.067} C_VEL
LIN {X 0,Y 171.82,Z 1105.966,A -85,B 0,C 180,E1 6326.338,E2 6326.338} C_VEL
LIN {X 0,Y 188.448,Z 1094.508,A -85,B 0,C 180,E1 6321.791,E2 6321.791} C_VEL
LIN {X 0,Y 205.201,Z 1081.967,A -85,B 0,C 180,E1 6318.161,E2 6318.161} C_VEL
LIN {X 0,Y 222.377,Z 1067.458,A -85,B 0,C 180,E1 6315.117,E2 6315.117} C_VEL
LIN {X 0,Y 238.811,Z 1052.137,A -85,B 0,C 180,E1 6312.692,E2 6312.692} C_VEL
LIN {X 0,Y 254.413,Z 1035.663,A -85,B 0,C 180,E1 6310.719,E2 6310.719} C_VEL
LIN {X 0,Y 269.815,Z 1017.509,A -85,B 0,C 180,E1 6309.028,E2 6309.028} C_VEL
LIN {X 0,Y 283.329,Z 999.297,A -85,B 0,C 180,E1 6307.707,E2 6307.707} C_VEL
LIN {X 0,Y 296.415,Z 979.42,A -85,B 0,C 180,E1 6306.568,E2 6306.568} C_VEL
LIN {X 0,Y 307.477,Z 959.891,A -85,B 0,C 180,E1 6305.678,E2 6305.678} C_VEL
LIN {X 0,Y 318.128,Z 938.303,A -85,B 0,C 180,E1 6304.896,E2 6304.896} C_VEL
LIN {X 0,Y 326.882,Z 916.887,A -85,B 0,C 180,E1 6304.291,E2 6304.291} C_VEL
LIN {X 0,Y 334.753,Z 893.814,A -85,B 0,C 180,E1 6303.777,E2 6303.777} C_VEL
LIN {X 0,Y 340.778,Z 870.851,A -85,B 0,C 180,E1 6303.388,E2 6303.388} C_VEL
LIN {X 0,Y 345.563,Z 846.366,A -85,B 0,C 180,E1 6303.051,E2 6303.051} C_VEL
LIN {X 0,Y 354.402,Z 773.857,A -85,B 0,C 180,E1 6302.161,E2 6302.161} C_VEL
LIN {X 0,Y 358.921,Z 735.863,A -85,B 0,C 180,E1 6301.676,E2 6301.676} C_VEL
LIN {X 0,Y 358.531,Z 734.494,A -85,B 0,C 180,E1 6299.361,E2 6299.361} C_VEL
LIN {X 0,Y 358.643,Z 736.427,A -85,B 0,C 180,E1 6295.523,E2 6295.523} C_VEL
LIN {X 0,Y 358.708,Z 737.233,A -85,B 0,C 180,E1 6295.028,E2 6295.028} C_VEL
LIN {X 0,Y 345.68,Z 845.639,A -85,B 0,C 180,E1 6293.743,E2 6293.743} C_VEL
LIN {X 0,Y 340.932,Z 870.389,A -85,B 0,C 180,E1 6293.415,E2 6293.415} C_VEL
LIN {X 0,Y 335.226,Z 892.349,A -85,B 0,C 180,E1 6293.06,E2 6293.06} C_VEL
LIN {X 0,Y 327.711,Z 914.865,A -85,B 0,C 180,E1 6292.579,E2 6292.579} C_VEL
LIN {X 0,Y 319.556,Z 935.103,A -85,B 0,C 180,E1 6292.027,E2 6292.027} C_VEL
LIN {X 0,Y 308.575,Z 957.875,A -85,B 0,C 180,E1 6291.231,E2 6291.231} C_VEL
LIN {X 0,Y 297.665,Z 977.258,A -85,B 0,C 180,E1 6290.369,E2 6290.369} C_VEL
LIN {X 0,Y 284.48,Z 997.473,A -85,B 0,C 180,E1 6289.233,E2 6289.233} C_VEL
LIN {X 0,Y 271.425,Z 1015.082,A -85,B 0,C 180,E1 6287.979,E2 6287.979} C_VEL
LIN {X 0,Y 255.774,Z 1033.595,A -85,B 0,C 180,E1 6286.278,E2 6286.278} C_VEL
LIN {X 0,Y 240.829,Z 1049.31,A -85,B 0,C 180,E1 6284.416,E2 6284.416} C_VEL
LIN {X 0,Y 223.973,Z 1064.969,A -85,B 0,C 180,E1 6281.973,E2 6281.973} C_VEL
LIN {X 0,Y 207.45,Z 1078.755,A -85,B 0,C 180,E1 6279.104,E2 6279.104} C_VEL
LIN {X 0,Y 190.186,Z 1091.489,A -85,B 0,C 180,E1 6275.442,E2 6275.442} C_VEL
LIN {X 0,Y 173.701,Z 1102.556,A -85,B 0,C 180,E1 6271.042,E2 6271.042} C_VEL
LIN {X 0,Y 157.702,Z 1112.096,A -85,B 0,C 180,E1 6265.513,E2 6265.513} C_VEL
LIN {X 0,Y 142.805,Z 1120.375,A -85,B 0,C 180,E1 6258.521,E2 6258.521} C_VEL
LIN {X 0,Y 130.307,Z 1126.751,A -85,B 0,C 180,E1 6250.133,E2 6250.133} C_VEL
LIN {X 0,Y 120.498,Z 1131.753,A -85,B 0,C 180,E1 6239.86,E2 6239.86} C_VEL
LIN {X 0,Y 114.844,Z 1134.745,A -85,B 0,C 180,E1 6229.32,E2 6229.32} C_VEL
LIN {X 0,Y 112.43,Z 1136.405,A -85,B 0,C 180,E1 6218.696,E2 6218.696} C_VEL
LIN {X 0,Y 112.063,Z 1136.821,A -85,B 0,C 180,E1 6209.489,E2 6209.489} C_VEL
LIN {X 0,Y 112.608,Z 1136.242,A -85,B 0,C 180,E1 6199.771,E2 6199.771} C_VEL
LIN {X 0,Y 115.227,Z 1134.559,A -85,B 0,C 180,E1 6189.584,E2 6189.584} C_VEL
LIN {X 0,Y 121.826,Z 1131.151,A -85,B 0,C 180,E1 6178.313,E2 6178.313} C_VEL
LIN {X 0,Y 131.709,Z 1126.124,A -85,B 0,C 180,E1 6168.664,E2 6168.664} C_VEL
LIN {X 0,Y 145.155,Z 1119.198,A -85,B 0,C 180,E1 6160.127,E2 6160.127} C_VEL
LIN {X 0,Y 159.003,Z 1111.484,A -85,B 0,C 180,E1 6153.892,E2 6153.892} C_VEL
LIN {X 0,Y 175.898,Z 1101.259,A -85,B 0,C 180,E1 6148.225,E2 6148.225} C_VEL
LIN {X 0,Y 191.718,Z 1090.606,A -85,B 0,C 180,E1 6144.118,E2 6144.118} C_VEL
LIN {X 0,Y 210.061,Z 1076.859,A -85,B 0,C 180,E1 6140.327,E2 6140.327} C_VEL
LIN {X 0,Y 225.647,Z 1063.775,A -85,B 0,C 180,E1 6137.69,E2 6137.69} C_VEL
LIN {X 0,Y 242.547,Z 1047.868,A -85,B 0,C 180,E1 6135.278,E2 6135.278} C_VEL
LIN {X 0,Y 257.08,Z 1032.503,A -85,B 0,C 180,E1 6133.495,E2 6133.495} C_VEL
LIN {X 0,Y 272.747,Z 1013.78,A -85,B 0,C 180,E1 6131.811,E2 6131.811} C_VEL
LIN {X 0,Y 285.352,Z 996.706,A -85,B 0,C 180,E1 6130.613,E2 6130.613} C_VEL
LIN {X 0,Y 299.022,Z 975.516,A -85,B 0,C 180,E1 6129.444,E2 6129.444} C_VEL
LIN {X 0,Y 309.468,Z 956.824,A -85,B 0,C 180,E1 6128.625,E2 6128.625} C_VEL
LIN {X 0,Y 320.457,Z 933.778,A -85,B 0,C 180,E1 6127.833,E2 6127.833} C_VEL
LIN {X 0,Y 328.62,Z 913.361,A -85,B 0,C 180,E1 6127.287,E2 6127.287} C_VEL
LIN {X 0,Y 336.449,Z 889.203,A -85,B 0,C 180,E1 6126.788,E2 6126.788} C_VEL
LIN {X 0,Y 342.001,Z 867.287,A -85,B 0,C 180,E1 6126.445,E2 6126.445} C_VEL
LIN {X 0,Y 346.476,Z 842.449,A -85,B 0,C 180,E1 6126.123,E2 6126.123} C_VEL
LIN {X 0,Y 359.075,Z 737.382,A -85,B 0,C 180,E1 6124.872,E2 6124.872} C_VEL
LIN {X 0,Y 358.832,Z 736.182,A -85,B 0,C 180,E1 6123.515,E2 6123.515} C_VEL
LIN {X 0,Y 358.841,Z 734.94,A -85,B 0,C 180,E1 6120.479,E2 6120.479} C_VEL
LIN {X 0,Y 359.207,Z 736.187,A -85,B 0,C 180,E1 6118.298,E2 6118.298} C_VEL
LIN {X 0,Y 346.073,Z 845.202,A -85,B 0,C 180,E1 6116.968,E2 6116.968} C_VEL
LIN {X 0,Y 341.275,Z 870.196,A -85,B 0,C 180,E1 6116.626,E2 6116.626} C_VEL
LIN {X 0,Y 335.443,Z 892.572,A -85,B 0,C 180,E1 6116.251,E2 6116.251} C_VEL
LIN {X 0,Y 327.864,Z 915.187,A -85,B 0,C 180,E1 6115.758,E2 6115.758} C_VEL
LIN {X 0,Y 319.589,Z 935.658,A -85,B 0,C 180,E1 6115.197,E2 6115.197} C_VEL
LIN {X 0,Y 309.089,Z 957.486,A -85,B 0,C 180,E1 6114.431,E2 6114.431} C_VEL
LIN {X 0,Y 298.341,Z 976.703,A -85,B 0,C 180,E1 6113.578,E2 6113.578} C_VEL
LIN {X 0,Y 284.803,Z 997.676,A -85,B 0,C 180,E1 6112.412,E2 6112.412} C_VEL
LIN {X 0,Y 280.202,Z 1003.985,A -85,B 0,C 180,E1 6112.21,E2 6112.21} C_VEL
LIN {X 0,Y 267.341,Z 1019.468,A -85,B 0,C 180,E1 6112.337,E2 6112.337} C_VEL
LIN {X 0,Y 262.36,Z 1025.136,A -85,B 0,C 180,E1 6112.076,E2 6112.076} C_VEL
LIN {X 0,Y 246.452,Z 1042.815,A -85,B 0,C 180,E1 6110.364,E2 6110.364} C_VEL
LIN {X 0,Y 229.766,Z 1059.075,A -85,B 0,C 180,E1 6108.281,E2 6108.281} C_VEL
LIN {X 0,Y 211.642,Z 1074.844,A -85,B 0,C 180,E1 6105.585,E2 6105.585} C_VEL
LIN {X 0,Y 195.797,Z 1087.118,A -85,B 0,C 180,E1 6102.74,E2 6102.74} C_VEL
LIN {X 0,Y 178.033,Z 1099.599,A -85,B 0,C 180,E1 6098.799,E2 6098.799} C_VEL
LIN {X 0,Y 161.262,Z 1110.126,A -85,B 0,C 180,E1 6094.035,E2 6094.035} C_VEL
LIN {X 0,Y 144.415,Z 1119.831,A -85,B 0,C 180,E1 6087.64,E2 6087.64} C_VEL
LIN {X 0,Y 130.273,Z 1127.315,A -85,B 0,C 180,E1 6080.133,E2 6080.133} C_VEL
LIN {X 0,Y 117.315,Z 1133.962,A -85,B 0,C 180,E1 6069.735,E2 6069.735} C_VEL
LIN {X 0,Y 109.64,Z 1138.016,A -85,B 0,C 180,E1 6059.503,E2 6059.503} C_VEL
LIN {X 0,Y 105.018,Z 1141.021,A -85,B 0,C 180,E1 6047.167,E2 6047.167} C_VEL
LIN {X 0,Y 103.998,Z 1142.241,A -85,B 0,C 180,E1 6036.071,E2 6036.071} C_VEL
LIN {X 0,Y 104.041,Z 1142.456,A -85,B 0,C 180,E1 6028.899,E2 6028.899} C_VEL
LIN {X 0,Y 104.1,Z 1141.95,A -85,B 0,C 180,E1 6020.044,E2 6020.044} C_VEL
LIN {X 0,Y 106.005,Z 1140.193,A -85,B 0,C 180,E1 6008.996,E2 6008.996} C_VEL
LIN {X 0,Y 111.173,Z 1137.133,A -85,B 0,C 180,E1 5997.951,E2 5997.951} C_VEL
LIN {X 0,Y 121.537,Z 1131.715,A -85,B 0,C 180,E1 5986.285,E2 5986.285} C_VEL
LIN {X 0,Y 133.524,Z 1125.54,A -85,B 0,C 180,E1 5977.883,E2 5977.883} C_VEL
LIN {X 0,Y 149.336,Z 1116.939,A -85,B 0,C 180,E1 5970.262,E2 5970.262} C_VEL
LIN {X 0,Y 164.358,Z 1108.112,A -85,B 0,C 180,E1 5964.979,E2 5964.979} C_VEL
LIN {X 0,Y 183.008,Z 1096.026,A -85,B 0,C 180,E1 5959.99,E2 5959.99} C_VEL
LIN {X 0,Y 199.268,Z 1084.337,A -85,B 0,C 180,E1 5956.583,E2 5956.583} C_VEL
LIN {X 0,Y 217.922,Z 1069.323,A -85,B 0,C 180,E1 5953.413,E2 5953.413} C_VEL
LIN {X 0,Y 233.44,Z 1055.374,A -85,B 0,C 180,E1 5951.222,E2 5951.222} C_VEL
LIN {X 0,Y 250.233,Z 1038.422,A -85,B 0,C 180,E1 5949.197,E2 5949.197} C_VEL
LIN {X 0,Y 264.631,Z 1022.073,A -85,B 0,C 180,E1 5947.688,E2 5947.688} C_VEL
LIN {X 0,Y 280.137,Z 1002.077,A -85,B 0,C 180,E1 5946.252,E2 5946.252} C_VEL
LIN {X 0,Y 292.685,Z 983.641,A -85,B 0,C 180,E1 5945.223,E2 5945.223} C_VEL
LIN {X 0,Y 305.317,Z 962.212,A -85,B 0,C 180,E1 5944.272,E2 5944.272} C_VEL
LIN {X 0,Y 315.089,Z 943.006,A -85,B 0,C 180,E1 5943.599,E2 5943.599} C_VEL
LIN {X 0,Y 324.901,Z 920.213,A -85,B 0,C 180,E1 5942.964,E2 5942.964} C_VEL
LIN {X 0,Y 332.481,Z 898.851,A -85,B 0,C 180,E1 5942.498,E2 5942.498} C_VEL
LIN {X 0,Y 339.502,Z 873.742,A -85,B 0,C 180,E1 5942.083,E2 5942.083} C_VEL
LIN {X 0,Y 344.225,Z 851.06,A -85,B 0,C 180,E1 5941.783,E2 5941.783} C_VEL
LIN {X 0,Y 348.798,Z 817.08,A -85,B 0,C 180,E1 5941.375,E2 5941.375} C_VEL
LIN {X 0,Y 357.689,Z 742.892,A -85,B 0,C 180,E1 5940.48,E2 5940.48} C_VEL
LIN {X 0,Y 357.497,Z 742.511,A -85,B 0,C 180,E1 5938.878,E2 5938.878} C_VEL
LIN {X 0,Y 357.521,Z 744.086,A -85,B 0,C 180,E1 5936.231,E2 5936.231} C_VEL
LIN {X 0,Y 345.101,Z 845.77,A -85,B 0,C 180,E1 5935.068,E2 5935.068} C_VEL
LIN {X 0,Y 340.325,Z 870.385,A -85,B 0,C 180,E1 5934.76,E2 5934.76} C_VEL
LIN {X 0,Y 334.547,Z 892.416,A -85,B 0,C 180,E1 5934.427,E2 5934.427} C_VEL
LIN {X 0,Y 326.776,Z 915.414,A -85,B 0,C 180,E1 5933.967,E2 5933.967} C_VEL
LIN {X 0,Y 318.546,Z 935.587,A -85,B 0,C 180,E1 5933.451,E2 5933.451} C_VEL
LIN {X 0,Y 307.601,Z 958,A -85,B 0,C 180,E1 5932.717,E2 5932.717} C_VEL
LIN {X 0,Y 296.428,Z 977.621,A -85,B 0,C 180,E1 5931.898,E2 5931.898} C_VEL
LIN {X 0,Y 283.088,Z 997.786,A -85,B 0,C 180,E1 5930.832,E2 5930.832} C_VEL
LIN {X 0,Y 270.052,Z 1015.134,A -85,B 0,C 180,E1 5929.67,E2 5929.67} C_VEL
LIN {X 0,Y 254.444,Z 1033.362,A -85,B 0,C 180,E1 5928.098,E2 5928.098} C_VEL
LIN {X 0,Y 239.695,Z 1048.653,A -85,B 0,C 180,E1 5926.401,E2 5926.401} C_VEL
LIN {X 0,Y 222.377,Z 1064.549,A -85,B 0,C 180,E1 5924.081,E2 5924.081} C_VEL
LIN {X 0,Y 206.582,Z 1077.488,A -85,B 0,C 180,E1 5921.564,E2 5921.564} C_VEL
LIN {X 0,Y 188.617,Z 1090.588,A -85,B 0,C 180,E1 5918.08,E2 5918.08} C_VEL
LIN {X 0,Y 172.272,Z 1101.263,A -85,B 0,C 180,E1 5914.112,E2 5914.112} C_VEL
LIN {X 0,Y 154.682,Z 1111.521,A -85,B 0,C 180,E1 5908.57,E2 5908.57} C_VEL
LIN {X 0,Y 140.109,Z 1119.256,A -85,B 0,C 180,E1 5902.388,E2 5902.388} C_VEL
LIN {X 0,Y 125.767,Z 1126.224,A -85,B 0,C 180,E1 5893.763,E2 5893.763} C_VEL
LIN {X 0,Y 115.429,Z 1131.071,A -85,B 0,C 180,E1 5884.267,E2 5884.267} C_VEL
LIN {X 0,Y 107.886,Z 1134.632,A -85,B 0,C 180,E1 5872.333,E2 5872.333} C_VEL
LIN {X 0,Y 104.797,Z 1136.357,A -85,B 0,C 180,E1 5861.558,E2 5861.558} C_VEL
LIN {X 0,Y 104.069,Z 1136.976,A -85,B 0,C 180,E1 5851.652,E2 5851.652} C_VEL
LIN {X 0,Y 104.323,Z 1136.756,A -85,B 0,C 180,E1 5842.289,E2 5842.289} C_VEL
LIN {X 0,Y 106.816,Z 1135.228,A -85,B 0,C 180,E1 5830.306,E2 5830.306} C_VEL
LIN {X 0,Y 112.406,Z 1132.501,A -85,B 0,C 180,E1 5819.533,E2 5819.533} C_VEL
LIN {X 0,Y 123.091,Z 1127.576,A -85,B 0,C 180,E1 5808.233,E2 5808.233} C_VEL
LIN {X 0,Y 135.564,Z 1121.615,A -85,B 0,C 180,E1 5799.907,E2 5799.907} C_VEL
LIN {X 0,Y 151.7,Z 1113.291,A -85,B 0,C 180,E1 5792.469,E2 5792.469} C_VEL
LIN {X 0,Y 166.68,Z 1104.795,A -85,B 0,C 180,E1 5787.397,E2 5787.397} C_VEL
LIN {X 0,Y 185.201,Z 1093.09,A -85,B 0,C 180,E1 5782.598,E2 5782.598} C_VEL
LIN {X 0,Y 201.298,Z 1081.727,A -85,B 0,C 180,E1 5779.304,E2 5779.304} C_VEL
LIN {X 0,Y 218.844,Z 1067.821,A -85,B 0,C 180,E1 5776.365,E2 5776.365} C_VEL
LIN {X 0,Y 234.149,Z 1054.243,A -85,B 0,C 180,E1 5774.218,E2 5774.218} C_VEL
LIN {X 0,Y 251.594,Z 1036.79,A -85,B 0,C 180,E1 5772.133,E2 5772.133} C_VEL
LIN {X 0,Y 265.574,Z 1020.993,A -85,B 0,C 180,E1 5770.681,E2 5770.681} C_VEL
LIN {X 0,Y 281.132,Z 1000.987,A -85,B 0,C 180,E1 5769.257,E2 5769.257} C_VEL
LIN {X 0,Y 293.508,Z 982.826,A -85,B 0,C 180,E1 5768.251,E2 5768.251} C_VEL
LIN {X 0,Y 305.991,Z 961.63,A -85,B 0,C 180,E1 5767.322,E2 5767.322} C_VEL
LIN {X 0,Y 315.602,Z 942.735,A -85,B 0,C 180,E1 5766.667,E2 5766.667} C_VEL
LIN {X 0,Y 325.278,Z 920.278,A -85,B 0,C 180,E1 5766.05,E2 5766.05} C_VEL
LIN {X 0,Y 332.7,Z 899.396,A -85,B 0,C 180,E1 5765.599,E2 5765.599} C_VEL
LIN {X 0,Y 339.798,Z 874.127,A -85,B 0,C 180,E1 5765.196,E2 5765.196} C_VEL
LIN {X 0,Y 344.509,Z 851.545,A -85,B 0,C 180,E1 5764.908,E2 5764.908} C_VEL
LIN {X 0,Y 349.092,Z 817.604,A -85,B 0,C 180,E1 5764.511,E2 5764.511} C_VEL
LIN {X 0,Y 357.872,Z 744.229,A -85,B 0,C 180,E1 5763.644,E2 5763.644} C_VEL
LIN {X 0,Y 357.865,Z 742.883,A -85,B 0,C 180,E1 5760.48,E2 5760.48} C_VEL
LIN {X 0,Y 357.964,Z 743.467,A -85,B 0,C 180,E1 5759.491,E2 5759.491} C_VEL
LIN {X 0,Y 345.493,Z 845.437,A -85,B 0,C 180,E1 5758.291,E2 5758.291} C_VEL
LIN {X 0,Y 340.648,Z 870.356,A -85,B 0,C 180,E1 5757.968,E2 5757.968} C_VEL
LIN {X 0,Y 334.724,Z 892.86,A -85,B 0,C 180,E1 5757.614,E2 5757.614} C_VEL
LIN {X 0,Y 326.873,Z 915.941,A -85,B 0,C 180,E1 5757.142,E2 5757.142} C_VEL
LIN {X 0,Y 318.215,Z 937.034,A -85,B 0,C 180,E1 5756.595,E2 5756.595} C_VEL
LIN {X 0,Y 307.76,Z 958.299,A -85,B 0,C 180,E1 5755.889,E2 5755.889} C_VEL
LIN {X 0,Y 296.767,Z 977.649,A -85,B 0,C 180,E1 5755.077,E2 5755.077} C_VEL
LIN {X 0,Y 282.908,Z 998.67,A -85,B 0,C 180,E1 5753.968,E2 5753.968} C_VEL
LIN {X 0,Y 270.088,Z 1015.779,A -85,B 0,C 180,E1 5752.823,E2 5752.823} C_VEL
LIN {X 0,Y 262.36,Z 1025.136,A -85,B 0,C 180,E1 5752.076,E2 5752.076} C_VEL
LIN {X 0,Y 257.27,Z 1030.919,A -85,B 0,C 180,E1 5751.793,E2 5751.793} C_VEL
LIN {X 0,Y 242.895,Z 1045.027,A -85,B 0,C 180,E1 5751.76,E2 5751.76} C_VEL
LIN {X 0,Y 237.436,Z 1050.246,A -85,B 0,C 180,E1 5751.402,E2 5751.402} C_VEL
LIN {X 0,Y 219.859,Z 1066.211,A -85,B 0,C 180,E1 5749.218,E2 5749.218} C_VEL
LIN {X 0,Y 203.374,Z 1079.58,A -85,B 0,C 180,E1 5746.774,E2 5746.774} C_VEL
LIN {X 0,Y 184.17,Z 1093.411,A -85,B 0,C 180,E1 5743.277,E2 5743.277} C_VEL
LIN {X 0,Y 166.792,Z 1104.616,A -85,B 0,C 180,E1 5739.26,E2 5739.26} C_VEL
LIN {X 0,Y 148.376,Z 1115.187,A -85,B 0,C 180,E1 5733.673,E2 5733.673} C_VEL
LIN {X 0,Y 132.371,Z 1123.595,A -85,B 0,C 180,E1 5726.978,E2 5726.978} C_VEL
LIN {X 0,Y 117.926,Z 1130.523,A -85,B 0,C 180,E1 5718.258,E2 5718.258} C_VEL
LIN {X 0,Y 107.035,Z 1135.674,A -85,B 0,C 180,E1 5708.065,E2 5708.065} C_VEL
LIN {X 0,Y 99.194,Z 1139.567,A -85,B 0,C 180,E1 5694.877,E2 5694.877} C_VEL
LIN {X 0,Y 96.432,Z 1141.395,A -85,B 0,C 180,E1 5683.797,E2 5683.797} C_VEL
LIN {X 0,Y 96,Z 1142.132,A -85,B 0,C 180,E1 5674.181,E2 5674.181} C_VEL
LIN {X 0,Y 96.02,Z 1142.198,A -85,B 0,C 180,E1 5667.613,E2 5667.613} C_VEL
LIN {X 0,Y 96.241,Z 1141.592,A -85,B 0,C 180,E1 5658.007,E2 5658.007} C_VEL
LIN {X 0,Y 98.614,Z 1139.859,A -85,B 0,C 180,E1 5646.706,E2 5646.706} C_VEL
LIN {X 0,Y 105.034,Z 1136.583,A -85,B 0,C 180,E1 5634.5,E2 5634.5} C_VEL
LIN {X 0,Y 116.245,Z 1131.234,A -85,B 0,C 180,E1 5623.018,E2 5623.018} C_VEL
LIN {X 0,Y 129.66,Z 1124.819,A -85,B 0,C 180,E1 5614.396,E2 5614.396} C_VEL
LIN {X 0,Y 146.083,Z 1116.299,A -85,B 0,C 180,E1 5607.15,E2 5607.15} C_VEL
LIN {X 0,Y 162.66,Z 1106.951,A -85,B 0,C 180,E1 5601.841,E2 5601.841} C_VEL
LIN {X 0,Y 181.208,Z 1095.211,A -85,B 0,C 180,E1 5597.33,E2 5597.33} C_VEL
LIN {X 0,Y 198.894,Z 1082.789,A -85,B 0,C 180,E1 5593.964,E2 5593.964} C_VEL
LIN {X 0,Y 217.079,Z 1068.297,A -85,B 0,C 180,E1 5591.154,E2 5591.154} C_VEL
LIN {X 0,Y 233.858,Z 1053.41,A -85,B 0,C 180,E1 5589.004,E2 5589.004} C_VEL
LIN {X 0,Y 250.271,Z 1036.841,A -85,B 0,C 180,E1 5587.207,E2 5587.207} C_VEL
LIN {X 0,Y 265.32,Z 1019.859,A -85,B 0,C 180,E1 5585.778,E2 5585.778} C_VEL
LIN {X 0,Y 279.853,Z 1001.084,A -85,B 0,C 180,E1 5584.549,E2 5584.549} C_VEL
LIN {X 0,Y 293.036,Z 981.818,A -85,B 0,C 180,E1 5583.562,E2 5583.562} C_VEL
LIN {X 0,Y 305.311,Z 960.904,A -85,B 0,C 180,E1 5582.714,E2 5582.714} C_VEL
LIN {X 0,Y 316.166,Z 939.527,A -85,B 0,C 180,E1 5582.034,E2 5582.034} C_VEL
LIN {X 0,Y 325.079,Z 918.364,A -85,B 0,C 180,E1 5581.509,E2 5581.509} C_VEL
LIN {X 0,Y 332.526,Z 897.316,A -85,B 0,C 180,E1 5581.09,E2 5581.09} C_VEL
LIN {X 0,Y 339.211,Z 873.221,A -85,B 0,C 180,E1 5580.724,E2 5580.724} C_VEL
LIN {X 0,Y 344.068,Z 849.902,A -85,B 0,C 180,E1 5580.435,E2 5580.435} C_VEL
LIN {X 0,Y 349.142,Z 811.543,A -85,B 0,C 180,E1 5579.996,E2 5579.996} C_VEL
LIN {X 0,Y 356.557,Z 750.379,A -85,B 0,C 180,E1 5579.277,E2 5579.277} C_VEL
LIN {X 0,Y 356.438,Z 751.326,A -85,B 0,C 180,E1 5577.437,E2 5577.437} C_VEL
LIN {X 0,Y 344.708,Z 845.901,A -85,B 0,C 180,E1 5576.397,E2 5576.397} C_VEL
LIN {X 0,Y 339.886,Z 870.459,A -85,B 0,C 180,E1 5576.107,E2 5576.107} C_VEL
LIN {X 0,Y 334.03,Z 892.585,A -85,B 0,C 180,E1 5575.796,E2 5575.796} C_VEL
LIN {X 0,Y 326.523,Z 914.687,A -85,B 0,C 180,E1 5575.389,E2 5575.389} C_VEL
LIN {X 0,Y 318.22,Z 934.948,A -85,B 0,C 180,E1 5574.913,E2 5574.913} C_VEL
LIN {X 0,Y 306.979,Z 957.86,A -85,B 0,C 180,E1 5574.22,E2 5574.22} C_VEL
LIN {X 0,Y 295.887,Z 977.178,A -85,B 0,C 180,E1 5573.474,E2 5573.474} C_VEL
LIN {X 0,Y 282.198,Z 997.713,A -85,B 0,C 180,E1 5572.467,E2 5572.467} C_VEL
LIN {X 0,Y 268.495,Z 1015.722,A -85,B 0,C 180,E1 5571.34,E2 5571.34} C_VEL
LIN {X 0,Y 252.901,Z 1033.63,A -85,B 0,C 180,E1 5569.889,E2 5569.889} C_VEL
LIN {X 0,Y 237.922,Z 1048.912,A -85,B 0,C 180,E1 5568.296,E2 5568.296} C_VEL
LIN {X 0,Y 219.859,Z 1065.152,A -85,B 0,C 180,E1 5566.052,E2 5566.052} C_VEL
LIN {X 0,Y 203.266,Z 1078.417,A -85,B 0,C 180,E1 5563.584,E2 5563.584} C_VEL
LIN {X 0,Y 184.869,Z 1091.382,A -85,B 0,C 180,E1 5560.238,E2 5560.238} C_VEL
LIN {X 0,Y 167.231,Z 1102.502,A -85,B 0,C 180,E1 5556.179,E2 5556.179} C_VEL
LIN {X 0,Y 149.823,Z 1112.14,A -85,B 0,C 180,E1 5550.959,E2 5550.959} C_VEL
LIN {X 0,Y 133.23,Z 1120.506,A -85,B 0,C 180,E1 5544.149,E2 5544.149} C_VEL
LIN {X 0,Y 118.866,Z 1126.935,A -85,B 0,C 180,E1 5535.644,E2 5535.644} C_VEL
LIN {X 0,Y 107.105,Z 1132.026,A -85,B 0,C 180,E1 5524.714,E2 5524.714} C_VEL
LIN {X 0,Y 99.945,Z 1135.062,A -85,B 0,C 180,E1 5512.965,E2 5512.965} C_VEL
LIN {X 0,Y 96.735,Z 1136.697,A -85,B 0,C 180,E1 5501.326,E2 5501.326} C_VEL
LIN {X 0,Y 96.071,Z 1137.23,A -85,B 0,C 180,E1 5490.596,E2 5490.596} C_VEL
LIN {X 0,Y 96.564,Z 1136.858,A -85,B 0,C 180,E1 5479.861,E2 5479.861} C_VEL
LIN {X 0,Y 99.678,Z 1135.223,A -85,B 0,C 180,E1 5467.593,E2 5467.593} C_VEL
LIN {X 0,Y 106.648,Z 1132.252,A -85,B 0,C 180,E1 5455.768,E2 5455.768} C_VEL
LIN {X 0,Y 118.238,Z 1127.296,A -85,B 0,C 180,E1 5444.736,E2 5444.736} C_VEL
LIN {X 0,Y 132.478,Z 1120.941,A -85,B 0,C 180,E1 5436.138,E2 5436.138} C_VEL
LIN {X 0,Y 148.984,Z 1112.712,A -85,B 0,C 180,E1 5429.251,E2 5429.251} C_VEL
LIN {X 0,Y 166.336,Z 1103.206,A -85,B 0,C 180,E1 5423.976,E2 5423.976} C_VEL
LIN {X 0,Y 183.935,Z 1092.182,A -85,B 0,C 180,E1 5419.873,E2 5419.873} C_VEL
LIN {X 0,Y 201.417,Z 1080.072,A -85,B 0,C 180,E1 5416.642,E2 5416.642} C_VEL
LIN {X 0,Y 218.746,Z 1066.342,A -85,B 0,C 180,E1 5414.02,E2 5414.02} C_VEL
LIN {X 0,Y 236.004,Z 1051.123,A -85,B 0,C 180,E1 5411.848,E2 5411.848} C_VEL
LIN {X 0,Y 252.374,Z 1034.541,A -85,B 0,C 180,E1 5410.085,E2 5410.085} C_VEL
LIN {X 0,Y 268.004,Z 1016.774,A -85,B 0,C 180,E1 5408.627,E2 5408.627} C_VEL
LIN {X 0,Y 281.87,Z 998.641,A -85,B 0,C 180,E1 5407.482,E2 5407.482} C_VEL
LIN {X 0,Y 295.362,Z 978.64,A -85,B 0,C 180,E1 5406.489,E2 5406.489} C_VEL
LIN {X 0,Y 306.848,Z 958.741,A -85,B 0,C 180,E1 5405.712,E2 5405.712} C_VEL
LIN {X 0,Y 317.697,Z 936.964,A -85,B 0,C 180,E1 5405.044,E2 5405.044} C_VEL
LIN {X 0,Y 326.489,Z 915.703,A -85,B 0,C 180,E1 5404.537,E2 5404.537} C_VEL
LIN {X 0,Y 334.43,Z 892.433,A -85,B 0,C 180,E1 5404.107,E2 5404.107} C_VEL
LIN {X 0,Y 340.291,Z 870.266,A -85,B 0,C 180,E1 5403.797,E2 5403.797} C_VEL
LIN {X 0,Y 345.185,Z 845.101,A -85,B 0,C 180,E1 5403.503,E2 5403.503} C_VEL
LIN {X 0,Y 356.785,Z 751.521,A -85,B 0,C 180,E1 5402.461,E2 5402.461} C_VEL
LIN {X 0,Y 356.85,Z 750.973,A -85,B 0,C 180,E1 5400.691,E2 5400.691} C_VEL
LIN {X 0,Y 345.081,Z 845.779,A -85,B 0,C 180,E1 5399.616,E2 5399.616} C_VEL
LIN {X 0,Y 340.229,Z 870.429,A -85,B 0,C 180,E1 5399.314,E2 5399.314} C_VEL
LIN {X 0,Y 334.299,Z 892.787,A -85,B 0,C 180,E1 5398.987,E2 5398.987} C_VEL
LIN {X 0,Y 326.569,Z 915.401,A -85,B 0,C 180,E1 5398.56,E2 5398.56} C_VEL
LIN {X 0,Y 318.146,Z 935.843,A -85,B 0,C 180,E1 5398.076,E2 5398.076} C_VEL
LIN {X 0,Y 307.085,Z 958.278,A -85,B 0,C 180,E1 5397.387,E2 5397.387} C_VEL
LIN {X 0,Y 295.98,Z 977.624,A -85,B 0,C 180,E1 5396.633,E2 5396.633} C_VEL
LIN {X 0,Y 282.293,Z 998.187,A -85,B 0,C 180,E1 5395.626,E2 5395.626} C_VEL
LIN {X 0,Y 269.187,Z 1015.485,A -85,B 0,C 180,E1 5394.553,E2 5394.553} C_VEL
LIN {X 0,Y 252.838,Z 1034.439,A -85,B 0,C 180,E1 5393.038,E2 5393.038} C_VEL
LIN {X 0,Y 237.436,Z 1050.246,A -85,B 0,C 180,E1 5391.402,E2 5391.402} C_VEL
LIN {X 0,Y 231.868,Z 1055.422,A -85,B 0,C 180,E1 5391.013,E2 5391.013} C_VEL
LIN {X 0,Y 216.245,Z 1068.079,A -85,B 0,C 180,E1 5390.769,E2 5390.769} C_VEL
LIN {X 0,Y 210.299,Z 1072.727,A -85,B 0,C 180,E1 5390.284,E2 5390.284} C_VEL
LIN {X 0,Y 192.452,Z 1086.01,A -85,B 0,C 180,E1 5387.624,E2 5387.624} C_VEL
LIN {X 0,Y 173.607,Z 1098.626,A -85,B 0,C 180,E1 5384.121,E2 5384.121} C_VEL
LIN {X 0,Y 155.548,Z 1109.21,A -85,B 0,C 180,E1 5379.804,E2 5379.804} C_VEL
LIN {X 0,Y 137.794,Z 1118.669,A -85,B 0,C 180,E1 5374.132,E2 5374.132} C_VEL
LIN {X 0,Y 120.996,Z 1126.567,A -85,B 0,C 180,E1 5366.58,E2 5366.58} C_VEL
LIN {X 0,Y 106.217,Z 1133.1,A -85,B 0,C 180,E1 5356.457,E2 5356.457} C_VEL
LIN {X 0,Y 96.041,Z 1137.417,A -85,B 0,C 180,E1 5344.933,E2 5344.933} C_VEL
LIN {X 0,Y 89.751,Z 1140.513,A -85,B 0,C 180,E1 5330.886,E2 5330.886} C_VEL
LIN {X 0,Y 88.017,Z 1141.82,A -85,B 0,C 180,E1 5317.179,E2 5317.179} C_VEL
LIN {X 0,Y 88.041,Z 1142.036,A -85,B 0,C 180,E1 5308.698,E2 5308.698} C_VEL
LIN {X 0,Y 88.163,Z 1141.597,A -85,B 0,C 180,E1 5298.883,E2 5298.883} C_VEL
LIN {X 0,Y 90.928,Z 1139.764,A -85,B 0,C 180,E1 5285.3,E2 5285.3} C_VEL
LIN {X 0,Y 97.609,Z 1136.7,A -85,B 0,C 180,E1 5272.815,E2 5272.815} C_VEL
LIN {X 0,Y 110.173,Z 1131.277,A -85,B 0,C 180,E1 5260.327,E2 5260.327} C_VEL
LIN {X 0,Y 123.751,Z 1125.222,A -85,B 0,C 180,E1 5251.963,E2 5251.963} C_VEL
LIN {X 0,Y 141.693,Z 1116.489,A -85,B 0,C 180,E1 5244.45,E2 5244.45} C_VEL
LIN {X 0,Y 158.064,Z 1107.661,A -85,B 0,C 180,E1 5239.514,E2 5239.514} C_VEL
LIN {X 0,Y 178.025,Z 1095.563,A -85,B 0,C 180,E1 5234.971,E2 5234.971} C_VEL
LIN {X 0,Y 195.191,Z 1083.867,A -85,B 0,C 180,E1 5231.923,E2 5231.923} C_VEL
LIN {X 0,Y 214.694,Z 1068.831,A -85,B 0,C 180,E1 5229.123,E2 5229.123} C_VEL
LIN {X 0,Y 230.8,Z 1054.868,A -85,B 0,C 180,E1 5227.208,E2 5227.208} C_VEL
LIN {X 0,Y 248.684,Z 1037.298,A -85,B 0,C 180,E1 5225.399,E2 5225.399} C_VEL
LIN {X 0,Y 263.645,Z 1020.695,A -85,B 0,C 180,E1 5224.092,E2 5224.092} C_VEL
LIN {X 0,Y 278.832,Z 1001.438,A -85,B 0,C 180,E1 5222.915,E2 5222.915} C_VEL
LIN {X 0,Y 291.653,Z 982.96,A -85,B 0,C 180,E1 5222.033,E2 5222.033} C_VEL
LIN {X 0,Y 304.537,Z 961.411,A -85,B 0,C 180,E1 5221.218,E2 5221.218} C_VEL
LIN {X 0,Y 314.986,Z 941.112,A -85,B 0,C 180,E1 5220.618,E2 5220.618} C_VEL
LIN {X 0,Y 324.467,Z 919.102,A -85,B 0,C 180,E1 5220.107,E2 5220.107} C_VEL
LIN {X 0,Y 331.969,Z 898.165,A -85,B 0,C 180,E1 5219.72,E2 5219.72} C_VEL
LIN {X 0,Y 338.891,Z 873.62,A -85,B 0,C 180,E1 5219.375,E2 5219.375} C_VEL
LIN {X 0,Y 343.693,Z 850.878,A -85,B 0,C 180,E1 5219.112,E2 5219.112} C_VEL
LIN {X 0,Y 348.456,Z 816.069,A -85,B 0,C 180,E1 5218.729,E2 5218.729} C_VEL
LIN {X 0,Y 352.326,Z 784.49,A -85,B 0,C 180,E1 5218.38,E2 5218.38} C_VEL
LIN {X 0,Y 344.301,Z 847.418,A -85,B 0,C 180,E1 5217.712,E2 5217.712} C_VEL
LIN {X 0,Y 339.419,Z 871.446,A -85,B 0,C 180,E1 5217.447,E2 5217.447} C_VEL
LIN {X 0,Y 333.13,Z 894.739,A -85,B 0,C 180,E1 5217.142,E2 5217.142} C_VEL
LIN {X 0,Y 325.486,Z 916.512,A -85,B 0,C 180,E1 5216.763,E2 5216.763} C_VEL
LIN {X 0,Y 316.139,Z 938.788,A -85,B 0,C 180,E1 5216.265,E2 5216.265} C_VEL
LIN {X 0,Y 305.346,Z 959.953,A -85,B 0,C 180,E1 5215.656,E2 5215.656} C_VEL
LIN {X 0,Y 293.133,Z 980.703,A -85,B 0,C 180,E1 5214.894,E2 5214.894} C_VEL
LIN {X 0,Y 280.004,Z 999.74,A -85,B 0,C 180,E1 5214.003,E2 5214.003} C_VEL
LIN {X 0,Y 265.511,Z 1018.343,A -85,B 0,C 180,E1 5212.896,E2 5212.896} C_VEL
LIN {X 0,Y 250.177,Z 1035.406,A -85,B 0,C 180,E1 5211.57,E2 5211.57} C_VEL
LIN {X 0,Y 233.584,Z 1051.876,A -85,B 0,C 180,E1 5209.917,E2 5209.917} C_VEL
LIN {X 0,Y 216.746,Z 1066.461,A -85,B 0,C 180,E1 5207.959,E2 5207.959} C_VEL
LIN {X 0,Y 198.394,Z 1080.667,A -85,B 0,C 180,E1 5205.392,E2 5205.392} C_VEL
